  LIN {X 14334.988,Y 2494.793,Z -328.660,A -89.99654,B 0.00000,C 180.00000} ; insert
  LIN {X 14334.988,Y 2494.793,Z -328.660,A -89.99654,B 0.00000,C 180.00000} ; release
  LIN {X 14334.988,Y 2494.793,Z -28.660,A -89.99654,B 0.00000,C 180.00000} ; retreat
  ; Step 1131, bar 1482
  LIN {X 14434.988,Y 2494.793,Z 907.454,A -89.99654,B 0.00000,C 180.00000} ; outside
  LIN {X 14434.988,Y 2494.793,Z -78.660,A -89.99654,B 0.00000,C 180.00000} ; preinsert
  LIN {X 14434.988,Y 2494.793,Z -328.660,A -89.99654,B 0.00000,C 180.00000} ; insert
  LIN {X 14434.988,Y 2494.793,Z -328.660,A -89.99654,B 0.00000,C 180.00000} ; release
  LIN {X 14434.988,Y 2494.793,Z -28.660,A -89.99654,B 0.00000,C 180.00000} ; retreat
  ; Step 1132, bar 1484
  LIN {X 14534.988,Y 2494.793,Z 907.454,A -89.99654,B 0.00000,C 180.00000} ; outside
  LIN {X 14534.988,Y 2494.793,Z -78.660,A -89.99654,B 0.00000,C 180.00000} ; preinsert
  LIN {X 14534.988,Y 2494.793,Z -328.660,A -89.99654,B 0.00000,C 180.00000} ; insert
  LIN {X 14534.988,Y 2494.793,Z -328.660,A -89.99654,B 0.00000,C 180.00000} ; release
  LIN {X 14534.988,Y 2494.793,Z -28.660,A -89.99654,B 0.00000,C 180.00000} ; retreat
  ; Step 1133, bar 1486
  LIN {X 14634.988,Y 2494.793,Z 907.454,A -89.99654,B 0.00000,C 180.00000} ; outside
  LIN {X 14634.988,Y 2494.793,Z -78.660,A -89.99654,B 0.00000,C 180.00000} ; preinsert
  LIN {X 14634.988,Y 2494.793,Z -328.660,A -89.99654,B 0.00000,C 180.00000} ; insert
  LIN {X 14634.988,Y 2494.793,Z -328.660,A -89.99654,B 0.00000,C 180.00000} ; release
  LIN {X 14634.988,Y 2494.793,Z -28.660,A -89.99654,B 0.00000,C 180.00000} ; retreat
  ; Step 1134, bar 1488
  LIN {X 14734.988,Y 2494.793,Z 907.454,A -89.99654,B 0.00000,C 180.00000} ; outside
  LIN {X 14734.988,Y 2494.793,Z -78.660,A -89.99654,B 0.00000,C 180.00000} ; preinsert
  LIN {X 14734.988,Y 2494.793,Z -328.660,A -89.99654,B 0.00000,C 180.00000} ; insert
  LIN {X 14734.988,Y 2494.793,Z -328.660,A -89.99654,B 0.00000,C 180.00000} ; release
  LIN {X 14734.988,Y 2494.793,Z -28.660,A -89.99654,B 0.00000,C 180.00000} ; retreat
  ; Step 1135, bar 1490
  LIN {X 14834.988,Y 2494.793,Z 907.454,A -89.99654,B 0.00000,C 180.00000} ; outside
  LIN {X 14834.988,Y 2494.793,Z -78.660,A -89.99654,B 0.00000,C 180.00000} ; preinsert
  LIN {X 14834.988,Y 2494.793,Z -328.660,A -89.99654,B 0.00000,C 180.00000} ; insert
  LIN {X 14834.988,Y 2494.793,Z -328.660,A -89.99654,B 0.00000,C 180.00000} ; release
  LIN {X 14834.988,Y 2494.793,Z -28.660,A -89.99654,B 0.00000,C 180.00000} ; retreat
  ; Step 1136, bar 1492
  LIN {X 14934.988,Y 2494.793,Z 907.454,A -89.99654,B 0.00000,C 180.00000} ; outside
  LIN {X 14934.988,Y 2494.793,Z -78.660,A -89.99654,B 0.00000,C 180.00000} ; preinsert
  LIN {X 14934.988,Y 2494.793,Z -328.660,A -89.99654,B 0.00000,C 180.00000} ; insert
  LIN {X 14934.988,Y 2494.793,Z -328.660,A -89.99654,B 0.00000,C 180.00000} ; release
  LIN {X 14934.988,Y 2494.793,Z -28.660,A -89.99654,B 0.00000,C 180.00000} ; retreat
  ; Step 1137, bar 1494
  LIN {X 15034.988,Y 2494.793,Z 907.454,A -89.99654,B 0.00000,C 180.00000} ; outside
  LIN {X 15034.988,Y 2494.793,Z -78.660,A -89.99654,B 0.00000,C 180.00000} ; preinsert
  LIN {X 15034.988,Y 2494.793,Z -328.660,A -89.99654,B 0.00000,C 180.00000} ; insert
  LIN {X 15034.988,Y 2494.793,Z -328.660,A -89.99654,B 0.00000,C 180.00000} ; release
  LIN {X 15034.988,Y 2494.793,Z -28.660,A -89.99654,B 0.00000,C 180.00000} ; retreat
  ; Step 1138, bar 1496
  LIN {X 15134.988,Y 2494.793,Z 907.454,A -89.99654,B 0.00000,C 180.00000} ; outside
  LIN {X 15134.988,Y 2494.793,Z -78.660,A -89.99654,B 0.00000,C 180.00000} ; preinsert
  LIN {X 15134.988,Y 2494.793,Z -328.660,A -89.99654,B 0.00000,C 180.00000} ; insert
  LIN {X 15134.988,Y 2494.793,Z -328.660,A -89.99654,B 0.00000,C 180.00000} ; release
  LIN {X 15134.988,Y 2494.793,Z -28.660,A -89.99654,B 0.00000,C 180.00000} ; retreat
  ; Step 1139, bar 1498
  LIN {X 15234.988,Y 2494.793,Z 907.454,A -89.99654,B 0.00000,C 180.00000} ; outside
  LIN {X 15234.988,Y 2494.793,Z -78.660,A -89.99654,B 0.00000,C 180.00000} ; preinsert
  LIN {X 15234.988,Y 2494.793,Z -328.660,A -89.99654,B 0.00000,C 180.00000} ; insert
  LIN {X 15234.988,Y 2494.793,Z -328.660,A -89.99654,B 0.00000,C 180.00000} ; release
  LIN {X 15234.988,Y 2494.793,Z -28.660,A -89.99654,B 0.00000,C 180.00000} ; retreat
  ; Step 1140, bar 1500
  LIN {X 15334.988,Y 2494.793,Z 907.454,A -89.99654,B 0.00000,C 180.00000} ; outside
  LIN {X 15334.988,Y 2494.793,Z -78.660,A -89.99654,B 0.00000,C 180.00000} ; preinsert
  LIN {X 15334.988,Y 2494.793,Z -328.660,A -89.99654,B 0.00000,C 180.00000} ; insert
  LIN {X 15334.988,Y 2494.793,Z -328.660,A -89.99654,B 0.00000,C 180.00000} ; release
  LIN {X 15334.988,Y 2494.793,Z -28.660,A -89.99654,B 0.00000,C 180.00000} ; retreat
  ; Step 1141, bar 1502
  LIN {X 15434.988,Y 2494.793,Z 907.454,A -89.99654,B 0.00000,C 180.00000} ; outside
  LIN {X 15434.988,Y 2494.793,Z -78.660,A -89.99654,B 0.00000,C 180.00000} ; preinsert
  LIN {X 15434.988,Y 2494.793,Z -328.660,A -89.99654,B 0.00000,C 180.00000} ; insert
  LIN {X 15434.988,Y 2494.793,Z -328.660,A -89.99654,B 0.00000,C 180.00000} ; release
  LIN {X 15434.988,Y 2494.793,Z -28.660,A -89.99654,B 0.00000,C 180.00000} ; retreat
  ; Step 1142, bar 1504
  LIN {X 15534.988,Y 2494.793,Z 907.454,A -89.99654,B 0.00000,C 180.00000} ; outside
  LIN {X 15534.988,Y 2494.793,Z -78.660,A -89.99654,B 0.00000,C 180.00000} ; preinsert
  LIN {X 15534.988,Y 2494.793,Z -328.660,A -89.99654,B 0.00000,C 180.00000} ; insert
  LIN {X 15534.988,Y 2494.793,Z -328.660,A -89.99654,B 0.00000,C 180.00000} ; release
  LIN {X 15534.988,Y 2494.793,Z -28.660,A -89.99654,B 0.00000,C 180.00000} ; retreat
  ; Step 1143, bar 1506
  LIN {X 15634.988,Y 2494.793,Z 907.454,A -89.99654,B 0.00000,C 180.00000} ; outside
  LIN {X 15634.988,Y 2494.793,Z -78.660,A -89.99654,B 0.00000,C 180.00000} ; preinsert
  LIN {X 15634.988,Y 2494.793,Z -328.660,A -89.99654,B 0.00000,C 180.00000} ; insert
  LIN {X 15634.988,Y 2494.793,Z -328.660,A -89.99654,B 0.00000,C 180.00000} ; release
  LIN {X 15634.988,Y 2494.793,Z -28.660,A -89.99654,B 0.00000,C 180.00000} ; retreat
  ; Step 1144, bar 1508
  LIN {X 15734.988,Y 2494.793,Z 907.454,A -89.99654,B 0.00000,C 180.00000} ; outside
  LIN {X 15734.988,Y 2494.793,Z -78.660,A -89.99654,B 0.00000,C 180.00000} ; preinsert
  LIN {X 15734.988,Y 2494.793,Z -328.660,A -89.99654,B 0.00000,C 180.00000} ; insert
  LIN {X 15734.988,Y 2494.793,Z -328.660,A -89.99654,B 0.00000,C 180.00000} ; release
  LIN {X 15734.988,Y 2494.793,Z -28.660,A -89.99654,B 0.00000,C 180.00000} ; retreat
  ; Step 1145, bar 1510
  LIN {X 15834.988,Y 2494.793,Z 907.454,A -89.99654,B 0.00000,C 180.00000} ; outside
  LIN {X 15834.988,Y 2494.793,Z -78.660,A -89.99654,B 0.00000,C 180.00000} ; preinsert
  LIN {X 15834.988,Y 2494.793,Z -328.660,A -89.99654,B 0.00000,C 180.00000} ; insert
  LIN {X 15834.988,Y 2494.793,Z -328.660,A -89.99654,B 0.00000,C 180.00000} ; release
  LIN {X 15834.988,Y 2494.793,Z -28.660,A -89.99654,B 0.00000,C 180.00000} ; retreat
  ; Step 1146, bar 1512
  LIN {X 15934.988,Y 2494.793,Z 907.454,A -89.99654,B 0.00000,C 180.00000} ; outside
  LIN {X 15934.988,Y 2494.793,Z -78.660,A -89.99654,B 0.00000,C 180.00000} ; preinsert
  LIN {X 15934.988,Y 2494.793,Z -328.660,A -89.99654,B 0.00000,C 180.00000} ; insert
  LIN {X 15934.988,Y 2494.793,Z -328.660,A -89.99654,B 0.00000,C 180.00000} ; release
  LIN {X 15934.988,Y 2494.793,Z -28.660,A -89.99654,B 0.00000,C 180.00000} ; retreat
  ; Step 1147, bar 1514
  LIN {X 16034.988,Y 2494.793,Z 907.454,A -89.99654,B 0.00000,C 180.00000} ; outside
  LIN {X 16034.988,Y 2494.793,Z -78.660,A -89.99654,B 0.00000,C 180.00000} ; preinsert
  LIN {X 16034.988,Y 2494.793,Z -328.660,A -89.99654,B 0.00000,C 180.00000} ; insert
  LIN {X 16034.988,Y 2494.793,Z -328.660,A -89.99654,B 0.00000,C 180.00000} ; release
  LIN {X 16034.988,Y 2494.793,Z -28.660,A -89.99654,B 0.00000,C 180.00000} ; retreat
  ; Step 1148, bar 1807
  LIN {X -14334.988,Y -2494.793,Z 907.454,A 90.00346,B 0.00000,C 180.00000} ; outside
  LIN {X -14334.988,Y -2494.793,Z -78.660,A 90.00346,B 0.00000,C 180.00000} ; preinsert
  LIN {X -14334.988,Y -2494.793,Z -328.660,A 90.00346,B 0.00000,C 180.00000} ; insert
  LIN {X -14334.988,Y -2494.793,Z -328.660,A 90.00346,B 0.00000,C 180.00000} ; release
  LIN {X -14334.988,Y -2494.793,Z -28.660,A 90.00346,B 0.00000,C 180.00000} ; retreat
  ; Step 1149, bar 1809
  LIN {X -14434.988,Y -2494.793,Z 907.454,A 90.00346,B 0.00000,C 180.00000} ; outside
  LIN {X -14434.988,Y -2494.793,Z -78.660,A 90.00346,B 0.00000,C 180.00000} ; preinsert
  LIN {X -14434.988,Y -2494.793,Z -328.660,A 90.00346,B 0.00000,C 180.00000} ; insert
  LIN {X -14434.988,Y -2494.793,Z -328.660,A 90.00346,B 0.00000,C 180.00000} ; release
  LIN {X -14434.988,Y -2494.793,Z -28.660,A 90.00346,B 0.00000,C 180.00000} ; retreat
  ; Step 1150, bar 1811
  LIN {X -14534.988,Y -2494.793,Z 907.454,A 90.00346,B 0.00000,C 180.00000} ; outside
  LIN {X -14534.988,Y -2494.793,Z -78.660,A 90.00346,B 0.00000,C 180.00000} ; preinsert
  LIN {X -14534.988,Y -2494.793,Z -328.660,A 90.00346,B 0.00000,C 180.00000} ; insert
  LIN {X -14534.988,Y -2494.793,Z -328.660,A 90.00346,B 0.00000,C 180.00000} ; release
  LIN {X -14534.988,Y -2494.793,Z -28.660,A 90.00346,B 0.00000,C 180.00000} ; retreat
  ; Step 1151, bar 1813
  LIN {X -14634.988,Y -2494.793,Z 907.454,A 90.00346,B 0.00000,C 180.00000} ; outside
  LIN {X -14634.988,Y -2494.793,Z -78.660,A 90.00346,B 0.00000,C 180.00000} ; preinsert
  LIN {X -14634.988,Y -2494.793,Z -328.660,A 90.00346,B 0.00000,C 180.00000} ; insert
  LIN {X -14634.988,Y -2494.793,Z -328.660,A 90.00346,B 0.00000,C 180.00000} ; release
  LIN {X -14634.988,Y -2494.793,Z -28.660,A 90.00346,B 0.00000,C 180.00000} ; retreat
  ; Step 1152, bar 1815
  LIN {X -14734.988,Y -2494.793,Z 907.454,A 90.00346,B 0.00000,C 180.00000} ; outside
  LIN {X -14734.988,Y -2494.793,Z -78.660,A 90.00346,B 0.00000,C 180.00000} ; preinsert
  LIN {X -14734.988,Y -2494.793,Z -328.660,A 90.00346,B 0.00000,C 180.00000} ; insert
  LIN {X -14734.988,Y -2494.793,Z -328.660,A 90.00346,B 0.00000,C 180.00000} ; release
  LIN {X -14734.988,Y -2494.793,Z -28.660,A 90.00346,B 0.00000,C 180.00000} ; retreat
  ; Step 1153, bar 1817
  LIN {X -14834.988,Y -2494.793,Z 907.454,A 90.00346,B 0.00000,C 180.00000} ; outside
  LIN {X -14834.988,Y -2494.793,Z -78.660,A 90.00346,B 0.00000,C 180.00000} ; preinsert
  LIN {X -14834.988,Y -2494.793,Z -328.660,A 90.00346,B 0.00000,C 180.00000} ; insert
  LIN {X -14834.988,Y -2494.793,Z -328.660,A 90.00346,B 0.00000,C 180.00000} ; release
  LIN {X -14834.988,Y -2494.793,Z -28.660,A 90.00346,B 0.00000,C 180.00000} ; retreat
  ; Step 1154, bar 1819
  LIN {X -14934.988,Y -2494.793,Z 907.454,A 90.00346,B 0.00000,C 180.00000} ; outside
  LIN {X -14934.988,Y -2494.793,Z -78.660,A 90.00346,B 0.00000,C 180.00000} ; preinsert
  LIN {X -14934.988,Y -2494.793,Z -328.660,A 90.00346,B 0.00000,C 180.00000} ; insert
  LIN {X -14934.988,Y -2494.793,Z -328.660,A 90.00346,B 0.00000,C 180.00000} ; release
  LIN {X -14934.988,Y -2494.793,Z -28.660,A 90.00346,B 0.00000,C 180.00000} ; retreat
  ; Step 1155, bar 1821
  LIN {X -15034.988,Y -2494.793,Z 907.454,A 90.00346,B 0.00000,C 180.00000} ; outside
  LIN {X -15034.988,Y -2494.793,Z -78.660,A 90.00346,B 0.00000,C 180.00000} ; preinsert
  LIN {X -15034.988,Y -2494.793,Z -328.660,A 90.00346,B 0.00000,C 180.00000} ; insert
  LIN {X -15034.988,Y -2494.793,Z -328.660,A 90.00346,B 0.00000,C 180.00000} ; release
  LIN {X -15034.988,Y -2494.793,Z -28.660,A 90.00346,B 0.00000,C 180.00000} ; retreat
  ; Step 1156, bar 1823
  LIN {X -15134.988,Y -2494.793,Z 907.454,A 90.00346,B 0.00000,C 180.00000} ; outside
  LIN {X -15134.988,Y -2494.793,Z -78.660,A 90.00346,B 0.00000,C 180.00000} ; preinsert
  LIN {X -15134.988,Y -2494.793,Z -328.660,A 90.00346,B 0.00000,C 180.00000} ; insert
  LIN {X -15134.988,Y -2494.793,Z -328.660,A 90.00346,B 0.00000,C 180.00000} ; release
  LIN {X -15134.988,Y -2494.793,Z -28.660,A 90.00346,B 0.00000,C 180.00000} ; retreat
  ; Step 1157, bar 1825
  LIN {X -15234.988,Y -2494.793,Z 907.454,A 90.00346,B 0.00000,C 180.00000} ; outside
  LIN {X -15234.988,Y -2494.793,Z -78.660,A 90.00346,B 0.00000,C 180.00000} ; preinsert
  LIN {X -15234.988,Y -2494.793,Z -328.660,A 90.00346,B 0.00000,C 180.00000} ; insert
  LIN {X -15234.988,Y -2494.793,Z -328.660,A 90.00346,B 0.00000,C 180.00000} ; release
  LIN {X -15234.988,Y -2494.793,Z -28.660,A 90.00346,B 0.00000,C 180.00000} ; retreat
  ; Step 1158, bar 1829
  LIN {X -15434.988,Y -2494.793,Z 907.454,A 90.00346,B 0.00000,C 180.00000} ; outside
  LIN {X -15434.988,Y -2494.793,Z -78.660,A 90.00346,B 0.00000,C 180.00000} ; preinsert
  LIN {X -15434.988,Y -2494.793,Z -328.660,A 90.00346,B 0.00000,C 180.00000} ; insert
  LIN {X -15434.988,Y -2494.793,Z -328.660,A 90.00346,B 0.00000,C 180.00000} ; release
  LIN {X -15434.988,Y -2494.793,Z -28.660,A 90.00346,B 0.00000,C 180.00000} ; retreat
  ; Step 1159, bar 1827
  LIN {X -15334.988,Y -2494.793,Z 907.454,A 90.00346,B 0.00000,C 180.00000} ; outside
  LIN {X -15334.988,Y -2494.793,Z -78.660,A 90.00346,B 0.00000,C 180.00000} ; preinsert
  LIN {X -15334.988,Y -2494.793,Z -328.660,A 90.00346,B 0.00000,C 180.00000} ; insert
  LIN {X -15334.988,Y -2494.793,Z -328.660,A 90.00346,B 0.00000,C 180.00000} ; release
  LIN {X -15334.988,Y -2494.793,Z -28.660,A 90.00346,B 0.00000,C 180.00000} ; retreat
  ; Step 1160, bar 1831
  LIN {X -15534.988,Y -2494.793,Z 907.454,A 90.00346,B 0.00000,C 180.00000} ; outside
  LIN {X -15534.988,Y -2494.793,Z -78.660,A 90.00346,B 0.00000,C 180.00000} ; preinsert
  LIN {X -15534.988,Y -2494.793,Z -328.660,A 90.00346,B 0.00000,C 180.00000} ; insert
  LIN {X -15534.988,Y -2494.793,Z -328.660,A 90.00346,B 0.00000,C 180.00000} ; release
  LIN {X -15534.988,Y -2494.793,Z -28.660,A 90.00346,B 0.00000,C 180.00000} ; retreat
  ; Step 1161, bar 1833
  LIN {X -15634.988,Y -2494.793,Z 907.454,A 90.00346,B 0.00000,C 180.00000} ; outside
  LIN {X -15634.988,Y -2494.793,Z -78.660,A 90.00346,B 0.00000,C 180.00000} ; preinsert
  LIN {X -15634.988,Y -2494.793,Z -328.660,A 90.00346,B 0.00000,C 180.00000} ; insert
  LIN {X -15634.988,Y -2494.793,Z -328.660,A 90.00346,B 0.00000,C 180.00000} ; release
  LIN {X -15634.988,Y -2494.793,Z -28.660,A 90.00346,B 0.00000,C 180.00000} ; retreat
  ; Step 1162, bar 1835
  LIN {X -15734.988,Y -2494.793,Z 907.454,A 90.00346,B 0.00000,C 180.00000} ; outside
  LIN {X -15734.988,Y -2494.793,Z -78.660,A 90.00346,B 0.00000,C 180.00000} ; preinsert
  LIN {X -15734.988,Y -2494.793,Z -328.660,A 90.00346,B 0.00000,C 180.00000} ; insert
  LIN {X -15734.988,Y -2494.793,Z -328.660,A 90.00346,B 0.00000,C 180.00000} ; release
  LIN {X -15734.988,Y -2494.793,Z -28.660,A 90.00346,B 0.00000,C 180.00000} ; retreat
  ; Step 1163, bar 1837
  LIN {X -15834.988,Y -2494.793,Z 907.454,A 90.00346,B 0.00000,C 180.00000} ; outside
  LIN {X -15834.988,Y -2494.793,Z -78.660,A 90.00346,B 0.00000,C 180.00000} ; preinsert
  LIN {X -15834.988,Y -2494.793,Z -328.660,A 90.00346,B 0.00000,C 180.00000} ; insert
  LIN {X -15834.988,Y -2494.793,Z -328.660,A 90.00346,B 0.00000,C 180.00000} ; release
  LIN {X -15834.988,Y -2494.793,Z -28.660,A 90.00346,B 0.00000,C 180.00000} ; retreat
  ; Step 1164, bar 1839
  LIN {X -15934.988,Y -2494.793,Z 907.454,A 90.00346,B 0.00000,C 180.00000} ; outside
  LIN {X -15934.988,Y -2494.793,Z -78.660,A 90.00346,B 0.00000,C 180.00000} ; preinsert
  LIN {X -15934.988,Y -2494.793,Z -328.660,A 90.00346,B 0.00000,C 180.00000} ; insert
  LIN {X -15934.988,Y -2494.793,Z -328.660,A 90.00346,B 0.00000,C 180.00000} ; release
  LIN {X -15934.988,Y -2494.793,Z -28.660,A 90.00346,B 0.00000,C 180.00000} ; retreat
  ; Step 1165, bar 1841
  LIN {X -16034.988,Y -2494.793,Z 907.454,A 90.00346,B 0.00000,C 180.00000} ; outside
  LIN {X -16034.988,Y -2494.793,Z -78.660,A 90.00346,B 0.00000,C 180.00000} ; preinsert
  LIN {X -16034.988,Y -2494.793,Z -328.660,A 90.00346,B 0.00000,C 180.00000} ; insert
  LIN {X -16034.988,Y -2494.793,Z -328.660,A 90.00346,B 0.00000,C 180.00000} ; release
  LIN {X -16034.988,Y -2494.793,Z -28.660,A 90.00346,B 0.00000,C 180.00000} ; retreat
  ; Step 1166, bar 1479
  LIN {X 14334.988,Y -2494.793,Z 907.454,A 89.99654,B 0.00000,C -180.00000} ; outside
  LIN {X 14334.988,Y -2494.793,Z -78.660,A 89.99654,B 0.00000,C -180.00000} ; preinsert
  LIN {X 14334.988,Y -2494.793,Z -328.660,A 89.99654,B 0.00000,C -180.00000} ; insert
  LIN {X 14334.988,Y -2494.793,Z -328.660,A 89.99654,B 0.00000,C -180.00000} ; release
  LIN {X 14334.988,Y -2494.793,Z -28.660,A 89.99654,B 0.00000,C -180.00000} ; retreat
  ; Step 1167, bar 1481
  LIN {X 14434.988,Y -2494.793,Z 907.454,A 89.99654,B 0.00000,C -180.00000} ; outside
  LIN {X 14434.988,Y -2494.793,Z -78.660,A 89.99654,B 0.00000,C -180.00000} ; preinsert
  LIN {X 14434.988,Y -2494.793,Z -328.660,A 89.99654,B 0.00000,C -180.00000} ; insert
  LIN {X 14434.988,Y -2494.793,Z -328.660,A 89.99654,B 0.00000,C -180.00000} ; release
  LIN {X 14434.988,Y -2494.793,Z -28.660,A 89.99654,B 0.00000,C -180.00000} ; retreat
  ; Step 1168, bar 1483
  LIN {X 14534.988,Y -2494.793,Z 907.454,A 89.99654,B 0.00000,C -180.00000} ; outside
  LIN {X 14534.988,Y -2494.793,Z -78.660,A 89.99654,B 0.00000,C -180.00000} ; preinsert
  LIN {X 14534.988,Y -2494.793,Z -328.660,A 89.99654,B 0.00000,C -180.00000} ; insert
  LIN {X 14534.988,Y -2494.793,Z -328.660,A 89.99654,B 0.00000,C -180.00000} ; release
  LIN {X 14534.988,Y -2494.793,Z -28.660,A 89.99654,B 0.00000,C -180.00000} ; retreat
  ; Step 1169, bar 1485
  LIN {X 14634.988,Y -2494.793,Z 907.454,A 89.99654,B 0.00000,C -180.00000} ; outside
  LIN {X 14634.988,Y -2494.793,Z -78.660,A 89.99654,B 0.00000,C -180.00000} ; preinsert
  LIN {X 14634.988,Y -2494.793,Z -328.660,A 89.99654,B 0.00000,C -180.00000} ; insert
  LIN {X 14634.988,Y -2494.793,Z -328.660,A 89.99654,B 0.00000,C -180.00000} ; release
  LIN {X 14634.988,Y -2494.793,Z -28.660,A 89.99654,B 0.00000,C -180.00000} ; retreat
  ; Step 1170, bar 1487
  LIN {X 14734.988,Y -2494.793,Z 907.454,A 89.99654,B 0.00000,C -180.00000} ; outside
  LIN {X 14734.988,Y -2494.793,Z -78.660,A 89.99654,B 0.00000,C -180.00000} ; preinsert
  LIN {X 14734.988,Y -2494.793,Z -328.660,A 89.99654,B 0.00000,C -180.00000} ; insert
  LIN {X 14734.988,Y -2494.793,Z -328.660,A 89.99654,B 0.00000,C -180.00000} ; release
  LIN {X 14734.988,Y -2494.793,Z -28.660,A 89.99654,B 0.00000,C -180.00000} ; retreat
  ; Step 1171, bar 1489
  LIN {X 14834.988,Y -2494.793,Z 907.454,A 89.99654,B 0.00000,C -180.00000} ; outside
  LIN {X 14834.988,Y -2494.793,Z -78.660,A 89.99654,B 0.00000,C -180.00000} ; preinsert
  LIN {X 14834.988,Y -2494.793,Z -328.660,A 89.99654,B 0.00000,C -180.00000} ; insert
  LIN {X 14834.988,Y -2494.793,Z -328.660,A 89.99654,B 0.00000,C -180.00000} ; release
  LIN {X 14834.988,Y -2494.793,Z -28.660,A 89.99654,B 0.00000,C -180.00000} ; retreat
  ; Step 1172, bar 1491
  LIN {X 14934.988,Y -2494.793,Z 907.454,A 89.99654,B 0.00000,C -180.00000} ; outside
  LIN {X 14934.988,Y -2494.793,Z -78.660,A 89.99654,B 0.00000,C -180.00000} ; preinsert
  LIN {X 14934.988,Y -2494.793,Z -328.660,A 89.99654,B 0.00000,C -180.00000} ; insert
  LIN {X 14934.988,Y -2494.793,Z -328.660,A 89.99654,B 0.00000,C -180.00000} ; release
  LIN {X 14934.988,Y -2494.793,Z -28.660,A 89.99654,B 0.00000,C -180.00000} ; retreat
  ; Step 1173, bar 1493
  LIN {X 15034.988,Y -2494.793,Z 907.454,A 89.99654,B 0.00000,C -180.00000} ; outside
  LIN {X 15034.988,Y -2494.793,Z -78.660,A 89.99654,B 0.00000,C -180.00000} ; preinsert
  LIN {X 15034.988,Y -2494.793,Z -328.660,A 89.99654,B 0.00000,C -180.00000} ; insert
  LIN {X 15034.988,Y -2494.793,Z -328.660,A 89.99654,B 0.00000,C -180.00000} ; release
  LIN {X 15034.988,Y -2494.793,Z -28.660,A 89.99654,B 0.00000,C -180.00000} ; retreat
  ; Step 1174, bar 1495
  LIN {X 15134.988,Y -2494.793,Z 907.454,A 89.99654,B 0.00000,C -180.00000} ; outside
  LIN {X 15134.988,Y -2494.793,Z -78.660,A 89.99654,B 0.00000,C -180.00000} ; preinsert
  LIN {X 15134.988,Y -2494.793,Z -328.660,A 89.99654,B 0.00000,C -180.00000} ; insert
  LIN {X 15134.988,Y -2494.793,Z -328.660,A 89.99654,B 0.00000,C -180.00000} ; release
  LIN {X 15134.988,Y -2494.793,Z -28.660,A 89.99654,B 0.00000,C -180.00000} ; retreat
  ; Step 1175, bar 1497
  LIN {X 15234.988,Y -2494.793,Z 907.454,A 89.99654,B 0.00000,C -180.00000} ; outside
  LIN {X 15234.988,Y -2494.793,Z -78.660,A 89.99654,B 0.00000,C -180.00000} ; preinsert
  LIN {X 15234.988,Y -2494.793,Z -328.660,A 89.99654,B 0.00000,C -180.00000} ; insert
  LIN {X 15234.988,Y -2494.793,Z -328.660,A 89.99654,B 0.00000,C -180.00000} ; release
  LIN {X 15234.988,Y -2494.793,Z -28.660,A 89.99654,B 0.00000,C -180.00000} ; retreat
  ; Step 1176, bar 1499
  LIN {X 15334.988,Y -2494.793,Z 907.454,A 89.99654,B 0.00000,C -180.00000} ; outside
  LIN {X 15334.988,Y -2494.793,Z -78.660,A 89.99654,B 0.00000,C -180.00000} ; preinsert
  LIN {X 15334.988,Y -2494.793,Z -328.660,A 89.99654,B 0.00000,C -180.00000} ; insert
  LIN {X 15334.988,Y -2494.793,Z -328.660,A 89.99654,B 0.00000,C -180.00000} ; release
  LIN {X 15334.988,Y -2494.793,Z -28.660,A 89.99654,B 0.00000,C -180.00000} ; retreat
  ; Step 1177, bar 1501
  LIN {X 15434.988,Y -2494.793,Z 907.454,A 89.99654,B 0.00000,C -180.00000} ; outside
  LIN {X 15434.988,Y -2494.793,Z -78.660,A 89.99654,B 0.00000,C -180.00000} ; preinsert
  LIN {X 15434.988,Y -2494.793,Z -328.660,A 89.99654,B 0.00000,C -180.00000} ; insert
  LIN {X 15434.988,Y -2494.793,Z -328.660,A 89.99654,B 0.00000,C -180.00000} ; release
  LIN {X 15434.988,Y -2494.793,Z -28.660,A 89.99654,B 0.00000,C -180.00000} ; retreat
  ; Step 1178, bar 1503
  LIN {X 15534.988,Y -2494.793,Z 907.454,A 89.99654,B 0.00000,C -180.00000} ; outside
  LIN {X 15534.988,Y -2494.793,Z -78.660,A 89.99654,B 0.00000,C -180.00000} ; preinsert
  LIN {X 15534.988,Y -2494.793,Z -328.660,A 89.99654,B 0.00000,C -180.00000} ; insert
  LIN {X 15534.988,Y -2494.793,Z -328.660,A 89.99654,B 0.00000,C -180.00000} ; release
  LIN {X 15534.988,Y -2494.793,Z -28.660,A 89.99654,B 0.00000,C -180.00000} ; retreat
  ; Step 1179, bar 1505
  LIN {X 15634.988,Y -2494.793,Z 907.454,A 89.99654,B 0.00000,C -180.00000} ; outside
  LIN {X 15634.988,Y -2494.793,Z -78.660,A 89.99654,B 0.00000,C -180.00000} ; preinsert
  LIN {X 15634.988,Y -2494.793,Z -328.660,A 89.99654,B 0.00000,C -180.00000} ; insert
  LIN {X 15634.988,Y -2494.793,Z -328.660,A 89.99654,B 0.00000,C -180.00000} ; release
  LIN {X 15634.988,Y -2494.793,Z -28.660,A 89.99654,B 0.00000,C -180.00000} ; retreat
  ; Step 1180, bar 1507
  LIN {X 15734.988,Y -2494.793,Z 907.454,A 89.99654,B 0.00000,C -180.00000} ; outside
  LIN {X 15734.988,Y -2494.793,Z -78.660,A 89.99654,B 0.00000,C -180.00000} ; preinsert
  LIN {X 15734.988,Y -2494.793,Z -328.660,A 89.99654,B 0.00000,C -180.00000} ; insert
  LIN {X 15734.988,Y -2494.793,Z -328.660,A 89.99654,B 0.00000,C -180.00000} ; release
  LIN {X 15734.988,Y -2494.793,Z -28.660,A 89.99654,B 0.00000,C -180.00000} ; retreat
  ; Step 1181, bar 1509
  LIN {X 15834.988,Y -2494.793,Z 907.454,A 89.99654,B 0.00000,C -180.00000} ; outside
  LIN {X 15834.988,Y -2494.793,Z -78.660,A 89.99654,B 0.00000,C -180.00000} ; preinsert
  LIN {X 15834.988,Y -2494.793,Z -328.660,A 89.99654,B 0.00000,C -180.00000} ; insert
  LIN {X 15834.988,Y -2494.793,Z -328.660,A 89.99654,B 0.00000,C -180.00000} ; release
  LIN {X 15834.988,Y -2494.793,Z -28.660,A 89.99654,B 0.00000,C -180.00000} ; retreat
  ; Step 1182, bar 1511
  LIN {X 15934.988,Y -2494.793,Z 907.454,A 89.99654,B 0.00000,C -180.00000} ; outside
  LIN {X 15934.988,Y -2494.793,Z -78.660,A 89.99654,B 0.00000,C -180.00000} ; preinsert
  LIN {X 15934.988,Y -2494.793,Z -328.660,A 89.99654,B 0.00000,C -180.00000} ; insert
  LIN {X 15934.988,Y -2494.793,Z -328.660,A 89.99654,B 0.00000,C -180.00000} ; release
  LIN {X 15934.988,Y -2494.793,Z -28.660,A 89.99654,B 0.00000,C -180.00000} ; retreat
  ; Step 1183, bar 1513
  LIN {X 16034.988,Y -2494.793,Z 907.454,A 89.99654,B 0.00000,C -180.00000} ; outside
  LIN {X 16034.988,Y -2494.793,Z -78.660,A 89.99654,B 0.00000,C -180.00000} ; preinsert
  LIN {X 16034.988,Y -2494.793,Z -328.660,A 89.99654,B 0.00000,C -180.00000} ; insert
  LIN {X 16034.988,Y -2494.793,Z -328.660,A 89.99654,B 0.00000,C -180.00000} ; release
  LIN {X 16034.988,Y -2494.793,Z -28.660,A 89.99654,B 0.00000,C -180.00000} ; retreat
  ; Step 1184, bar 1808
  LIN {X -14334.988,Y 2494.793,Z 907.454,A -90.00346,B 0.00000,C -180.00000} ; outside
  LIN {X -14334.988,Y 2494.793,Z -78.660,A -90.00346,B 0.00000,C -180.00000} ; preinsert
  LIN {X -14334.988,Y 2494.793,Z -328.660,A -90.00346,B 0.00000,C -180.00000} ; insert
  LIN {X -14334.988,Y 2494.793,Z -328.660,A -90.00346,B 0.00000,C -180.00000} ; release
  LIN {X -14334.988,Y 2494.793,Z -28.660,A -90.00346,B 0.00000,C -180.00000} ; retreat
  ; Step 1185, bar 1810
  LIN {X -14434.988,Y 2494.793,Z 907.454,A -90.00346,B 0.00000,C -180.00000} ; outside
  LIN {X -14434.988,Y 2494.793,Z -78.660,A -90.00346,B 0.00000,C -180.00000} ; preinsert
  LIN {X -14434.988,Y 2494.793,Z -328.660,A -90.00346,B 0.00000,C -180.00000} ; insert
  LIN {X -14434.988,Y 2494.793,Z -328.660,A -90.00346,B 0.00000,C -180.00000} ; release
  LIN {X -14434.988,Y 2494.793,Z -28.660,A -90.00346,B 0.00000,C -180.00000} ; retreat
  ; Step 1186, bar 1812
  LIN {X -14534.988,Y 2494.793,Z 907.454,A -90.00346,B 0.00000,C -180.00000} ; outside
  LIN {X -14534.988,Y 2494.793,Z -78.660,A -90.00346,B 0.00000,C -180.00000} ; preinsert
  LIN {X -14534.988,Y 2494.793,Z -328.660,A -90.00346,B 0.00000,C -180.00000} ; insert
  LIN {X -14534.988,Y 2494.793,Z -328.660,A -90.00346,B 0.00000,C -180.00000} ; release
  LIN {X -14534.988,Y 2494.793,Z -28.660,A -90.00346,B 0.00000,C -180.00000} ; retreat
  ; Step 1187, bar 1814
  LIN {X -14634.988,Y 2494.793,Z 907.454,A -90.00346,B 0.00000,C -180.00000} ; outside
  LIN {X -14634.988,Y 2494.793,Z -78.660,A -90.00346,B 0.00000,C -180.00000} ; preinsert
  LIN {X -14634.988,Y 2494.793,Z -328.660,A -90.00346,B 0.00000,C -180.00000} ; insert
  LIN {X -14634.988,Y 2494.793,Z -328.660,A -90.00346,B 0.00000,C -180.00000} ; release
  LIN {X -14634.988,Y 2494.793,Z -28.660,A -90.00346,B 0.00000,C -180.00000} ; retreat
  ; Step 1188, bar 1816
  LIN {X -14734.988,Y 2494.793,Z 907.454,A -90.00346,B 0.00000,C -180.00000} ; outside
  LIN {X -14734.988,Y 2494.793,Z -78.660,A -90.00346,B 0.00000,C -180.00000} ; preinsert
  LIN {X -14734.988,Y 2494.793,Z -328.660,A -90.00346,B 0.00000,C -180.00000} ; insert
  LIN {X -14734.988,Y 2494.793,Z -328.660,A -90.00346,B 0.00000,C -180.00000} ; release
  LIN {X -14734.988,Y 2494.793,Z -28.660,A -90.00346,B 0.00000,C -180.00000} ; retreat
  ; Step 1189, bar 1818
  LIN {X -14834.988,Y 2494.793,Z 907.454,A -90.00346,B 0.00000,C -180.00000} ; outside
  LIN {X -14834.988,Y 2494.793,Z -78.660,A -90.00346,B 0.00000,C -180.00000} ; preinsert
  LIN {X -14834.988,Y 2494.793,Z -328.660,A -90.00346,B 0.00000,C -180.00000} ; insert
  LIN {X -14834.988,Y 2494.793,Z -328.660,A -90.00346,B 0.00000,C -180.00000} ; release
  LIN {X -14834.988,Y 2494.793,Z -28.660,A -90.00346,B 0.00000,C -180.00000} ; retreat
  ; Step 1190, bar 1820
  LIN {X -14934.988,Y 2494.793,Z 907.454,A -90.00346,B 0.00000,C -180.00000} ; outside
  LIN {X -14934.988,Y 2494.793,Z -78.660,A -90.00346,B 0.00000,C -180.00000} ; preinsert
  LIN {X -14934.988,Y 2494.793,Z -328.660,A -90.00346,B 0.00000,C -180.00000} ; insert
  LIN {X -14934.988,Y 2494.793,Z -328.660,A -90.00346,B 0.00000,C -180.00000} ; release
  LIN {X -14934.988,Y 2494.793,Z -28.660,A -90.00346,B 0.00000,C -180.00000} ; retreat
  ; Step 1191, bar 1822
  LIN {X -15034.988,Y 2494.793,Z 907.454,A -90.00346,B 0.00000,C -180.00000} ; outside
  LIN {X -15034.988,Y 2494.793,Z -78.660,A -90.00346,B 0.00000,C -180.00000} ; preinsert
  LIN {X -15034.988,Y 2494.793,Z -328.660,A -90.00346,B 0.00000,C -180.00000} ; insert
  LIN {X -15034.988,Y 2494.793,Z -328.660,A -90.00346,B 0.00000,C -180.00000} ; release
  LIN {X -15034.988,Y 2494.793,Z -28.660,A -90.00346,B 0.00000,C -180.00000} ; retreat
  ; Step 1192, bar 1824
  LIN {X -15134.988,Y 2494.793,Z 907.454,A -90.00346,B 0.00000,C -180.00000} ; outside
  LIN {X -15134.988,Y 2494.793,Z -78.660,A -90.00346,B 0.00000,C -180.00000} ; preinsert
  LIN {X -15134.988,Y 2494.793,Z -328.660,A -90.00346,B 0.00000,C -180.00000} ; insert
  LIN {X -15134.988,Y 2494.793,Z -328.660,A -90.00346,B 0.00000,C -180.00000} ; release
  LIN {X -15134.988,Y 2494.793,Z -28.660,A -90.00346,B 0.00000,C -180.00000} ; retreat
  ; Step 1193, bar 1826
  LIN {X -15234.988,Y 2494.793,Z 907.454,A -90.00346,B 0.00000,C -180.00000} ; outside
  LIN {X -15234.988,Y 2494.793,Z -78.660,A -90.00346,B 0.00000,C -180.00000} ; preinsert
  LIN {X -15234.988,Y 2494.793,Z -328.660,A -90.00346,B 0.00000,C -180.00000} ; insert
  LIN {X -15234.988,Y 2494.793,Z -328.660,A -90.00346,B 0.00000,C -180.00000} ; release
  LIN {X -15234.988,Y 2494.793,Z -28.660,A -90.00346,B 0.00000,C -180.00000} ; retreat
  ; Step 1194, bar 1830
  LIN {X -15434.988,Y 2494.793,Z 907.454,A -90.00346,B 0.00000,C -180.00000} ; outside
  LIN {X -15434.988,Y 2494.793,Z -78.660,A -90.00346,B 0.00000,C -180.00000} ; preinsert
  LIN {X -15434.988,Y 2494.793,Z -328.660,A -90.00346,B 0.00000,C -180.00000} ; insert
  LIN {X -15434.988,Y 2494.793,Z -328.660,A -90.00346,B 0.00000,C -180.00000} ; release
  LIN {X -15434.988,Y 2494.793,Z -28.660,A -90.00346,B 0.00000,C -180.00000} ; retreat
  ; Step 1195, bar 1828
  LIN {X -15334.988,Y 2494.793,Z 907.454,A -90.00346,B 0.00000,C -180.00000} ; outside
  LIN {X -15334.988,Y 2494.793,Z -78.660,A -90.00346,B 0.00000,C -180.00000} ; preinsert
  LIN {X -15334.988,Y 2494.793,Z -328.660,A -90.00346,B 0.00000,C -180.00000} ; insert
  LIN {X -15334.988,Y 2494.793,Z -328.660,A -90.00346,B 0.00000,C -180.00000} ; release
  LIN {X -15334.988,Y 2494.793,Z -28.660,A -90.00346,B 0.00000,C -180.00000} ; retreat
  ; Step 1196, bar 1832
  LIN {X -15534.988,Y 2494.793,Z 907.454,A -90.00346,B 0.00000,C -180.00000} ; outside
  LIN {X -15534.988,Y 2494.793,Z -78.660,A -90.00346,B 0.00000,C -180.00000} ; preinsert
  LIN {X -15534.988,Y 2494.793,Z -328.660,A -90.00346,B 0.00000,C -180.00000} ; insert
  LIN {X -15534.988,Y 2494.793,Z -328.660,A -90.00346,B 0.00000,C -180.00000} ; release
  LIN {X -15534.988,Y 2494.793,Z -28.660,A -90.00346,B 0.00000,C -180.00000} ; retreat
  ; Step 1197, bar 1834
  LIN {X -15634.988,Y 2494.793,Z 907.454,A -90.00346,B 0.00000,C -180.00000} ; outside
  LIN {X -15634.988,Y 2494.793,Z -78.660,A -90.00346,B 0.00000,C -180.00000} ; preinsert
  LIN {X -15634.988,Y 2494.793,Z -328.660,A -90.00346,B 0.00000,C -180.00000} ; insert
  LIN {X -15634.988,Y 2494.793,Z -328.660,A -90.00346,B 0.00000,C -180.00000} ; release
  LIN {X -15634.988,Y 2494.793,Z -28.660,A -90.00346,B 0.00000,C -180.00000} ; retreat
  ; Step 1198, bar 1836
  LIN {X -15734.988,Y 2494.793,Z 907.454,A -90.00346,B 0.00000,C -180.00000} ; outside
  LIN {X -15734.988,Y 2494.793,Z -78.660,A -90.00346,B 0.00000,C -180.00000} ; preinsert
  LIN {X -15734.988,Y 2494.793,Z -328.660,A -90.00346,B 0.00000,C -180.00000} ; insert
  LIN {X -15734.988,Y 2494.793,Z -328.660,A -90.00346,B 0.00000,C -180.00000} ; release
  LIN {X -15734.988,Y 2494.793,Z -28.660,A -90.00346,B 0.00000,C -180.00000} ; retreat
  ; Step 1199, bar 1838
  LIN {X -15834.988,Y 2494.793,Z 907.454,A -90.00346,B 0.00000,C -180.00000} ; outside
  LIN {X -15834.988,Y 2494.793,Z -78.660,A -90.00346,B 0.00000,C -180.00000} ; preinsert
  LIN {X -15834.988,Y 2494.793,Z -328.660,A -90.00346,B 0.00000,C -180.00000} ; insert
  LIN {X -15834.988,Y 2494.793,Z -328.660,A -90.00346,B 0.00000,C -180.00000} ; release
  LIN {X -15834.988,Y 2494.793,Z -28.660,A -90.00346,B 0.00000,C -180.00000} ; retreat
  ; Step 1200, bar 1840
  LIN {X -15934.988,Y 2494.793,Z 907.454,A -90.00346,B 0.00000,C -180.00000} ; outside
  LIN {X -15934.988,Y 2494.793,Z -78.660,A -90.00346,B 0.00000,C -180.00000} ; preinsert
  LIN {X -15934.988,Y 2494.793,Z -328.660,A -90.00346,B 0.00000,C -180.00000} ; insert
  LIN {X -15934.988,Y 2494.793,Z -328.660,A -90.00346,B 0.00000,C -180.00000} ; release
  LIN {X -15934.988,Y 2494.793,Z -28.660,A -90.00346,B 0.00000,C -180.00000} ; retreat
  ; Step 1201, bar 1842
  LIN {X -16034.988,Y 2494.793,Z 907.454,A -90.00346,B 0.00000,C -180.00000} ; outside
  LIN {X -16034.988,Y 2494.793,Z -78.660,A -90.00346,B 0.00000,C -180.00000} ; preinsert
  LIN {X -16034.988,Y 2494.793,Z -328.660,A -90.00346,B 0.00000,C -180.00000} ; insert
  LIN {X -16034.988,Y 2494.793,Z -328.660,A -90.00346,B 0.00000,C -180.00000} ; release
  LIN {X -16034.988,Y 2494.793,Z -28.660,A -90.00346,B 0.00000,C -180.00000} ; retreat
  ; Step 1202, bar 1515
  LIN {X 16134.974,Y -2655.018,Z 888.947,A 90.01124,B 0.00000,C 180.00000} ; outside
  LIN {X 16134.974,Y -2655.018,Z -60.206,A 90.01124,B 0.00000,C 180.00000} ; preinsert
  LIN {X 16134.974,Y -2655.018,Z -310.206,A 90.01124,B 0.00000,C 180.00000} ; insert
  LIN {X 16134.974,Y -2655.018,Z -310.206,A 90.01124,B 0.00000,C 180.00000} ; release
  LIN {X 16134.974,Y -2655.018,Z -10.206,A 90.01124,B 0.00000,C 180.00000} ; retreat
  ; Step 1203, bar 1517
  LIN {X 16234.974,Y -2655.018,Z 888.947,A 90.01124,B 0.00000,C 180.00000} ; outside
  LIN {X 16234.974,Y -2655.018,Z -60.206,A 90.01124,B 0.00000,C 180.00000} ; preinsert
  LIN {X 16234.974,Y -2655.018,Z -310.206,A 90.01124,B 0.00000,C 180.00000} ; insert
  LIN {X 16234.974,Y -2655.018,Z -310.206,A 90.01124,B 0.00000,C 180.00000} ; release
  LIN {X 16234.974,Y -2655.018,Z -10.206,A 90.01124,B 0.00000,C 180.00000} ; retreat
  ; Step 1204, bar 1844
  LIN {X -16134.974,Y 2655.018,Z 888.947,A -89.98876,B 0.00000,C 180.00000} ; outside
  LIN {X -16134.974,Y 2655.018,Z -60.206,A -89.98876,B 0.00000,C 180.00000} ; preinsert
  LIN {X -16134.974,Y 2655.018,Z -310.206,A -89.98876,B 0.00000,C 180.00000} ; insert
  LIN {X -16134.974,Y 2655.018,Z -310.206,A -89.98876,B 0.00000,C 180.00000} ; release
  LIN {X -16134.974,Y 2655.018,Z -10.206,A -89.98876,B 0.00000,C 180.00000} ; retreat
  ; Step 1205, bar 1846
  LIN {X -16234.974,Y 2655.018,Z 888.947,A -89.98876,B 0.00000,C 180.00000} ; outside
  LIN {X -16234.974,Y 2655.018,Z -60.206,A -89.98876,B 0.00000,C 180.00000} ; preinsert
  LIN {X -16234.974,Y 2655.018,Z -310.206,A -89.98876,B 0.00000,C 180.00000} ; insert
  LIN {X -16234.974,Y 2655.018,Z -310.206,A -89.98876,B 0.00000,C 180.00000} ; release
  LIN {X -16234.974,Y 2655.018,Z -10.206,A -89.98876,B 0.00000,C 180.00000} ; retreat
  ; Step 1206, bar 1516
  LIN {X 16134.974,Y 2655.018,Z 888.947,A -90.01124,B 0.00000,C -180.00000} ; outside
  LIN {X 16134.974,Y 2655.018,Z -60.206,A -90.01124,B 0.00000,C -180.00000} ; preinsert
  LIN {X 16134.974,Y 2655.018,Z -310.206,A -90.01124,B 0.00000,C -180.00000} ; insert
  LIN {X 16134.974,Y 2655.018,Z -310.206,A -90.01124,B 0.00000,C -180.00000} ; release
  LIN {X 16134.974,Y 2655.018,Z -10.206,A -90.01124,B 0.00000,C -180.00000} ; retreat
  ; Step 1207, bar 1518
  LIN {X 16234.974,Y 2655.018,Z 888.947,A -90.01124,B 0.00000,C -180.00000} ; outside
  LIN {X 16234.974,Y 2655.018,Z -60.206,A -90.01124,B 0.00000,C -180.00000} ; preinsert
  LIN {X 16234.974,Y 2655.018,Z -310.206,A -90.01124,B 0.00000,C -180.00000} ; insert
  LIN {X 16234.974,Y 2655.018,Z -310.206,A -90.01124,B 0.00000,C -180.00000} ; release
  LIN {X 16234.974,Y 2655.018,Z -10.206,A -90.01124,B 0.00000,C -180.00000} ; retreat
  ; Step 1208, bar 1843
  LIN {X -16134.974,Y -2655.018,Z 888.947,A 89.98876,B 0.00000,C 180.00000} ; outside
  LIN {X -16134.974,Y -2655.018,Z -60.206,A 89.98876,B 0.00000,C 180.00000} ; preinsert
  LIN {X -16134.974,Y -2655.018,Z -310.206,A 89.98876,B 0.00000,C 180.00000} ; insert
  LIN {X -16134.974,Y -2655.018,Z -310.206,A 89.98876,B 0.00000,C 180.00000} ; release
  LIN {X -16134.974,Y -2655.018,Z -10.206,A 89.98876,B 0.00000,C 180.00000} ; retreat
  ; Step 1209, bar 1845
  LIN {X -16234.974,Y -2655.018,Z 888.947,A 89.98876,B 0.00000,C 180.00000} ; outside
  LIN {X -16234.974,Y -2655.018,Z -60.206,A 89.98876,B 0.00000,C 180.00000} ; preinsert
  LIN {X -16234.974,Y -2655.018,Z -310.206,A 89.98876,B 0.00000,C 180.00000} ; insert
  LIN {X -16234.974,Y -2655.018,Z -310.206,A 89.98876,B 0.00000,C 180.00000} ; release
  LIN {X -16234.974,Y -2655.018,Z -10.206,A 89.98876,B 0.00000,C 180.00000} ; retreat
  ; Step 1210, bar 1520
  LIN {X 1986.078,Y 2753.934,Z 892.365,A -89.99242,B 0.00000,C 180.00000} ; outside
  LIN {X 1986.078,Y 2753.934,Z -48.972,A -89.99242,B 0.00000,C 180.00000} ; preinsert
  LIN {X 1986.078,Y 2753.934,Z -298.972,A -89.99242,B 0.00000,C 180.00000} ; insert
  LIN {X 1986.078,Y 2753.934,Z -298.972,A -89.99242,B 0.00000,C 180.00000} ; release
  LIN {X 1986.078,Y 2753.934,Z 1.028,A -89.99242,B 0.00000,C 180.00000} ; retreat
  ; Step 1211, bar 1522
  LIN {X 5986.078,Y 2753.934,Z 892.365,A -89.99242,B 0.00000,C 180.00000} ; outside
  LIN {X 5986.078,Y 2753.934,Z -48.972,A -89.99242,B 0.00000,C 180.00000} ; preinsert
  LIN {X 5986.078,Y 2753.934,Z -298.972,A -89.99242,B 0.00000,C 180.00000} ; insert
  LIN {X 5986.078,Y 2753.934,Z -298.972,A -89.99242,B 0.00000,C 180.00000} ; release
  LIN {X 5986.078,Y 2753.934,Z 1.028,A -89.99242,B 0.00000,C 180.00000} ; retreat
  ; Step 1212, bar 1524
  LIN {X 9986.078,Y 2753.934,Z 892.365,A -89.99242,B 0.00000,C 180.00000} ; outside
  LIN {X 9986.078,Y 2753.934,Z -48.972,A -89.99242,B 0.00000,C 180.00000} ; preinsert
  LIN {X 9986.078,Y 2753.934,Z -298.972,A -89.99242,B 0.00000,C 180.00000} ; insert
  LIN {X 9986.078,Y 2753.934,Z -298.972,A -89.99242,B 0.00000,C 180.00000} ; release
  LIN {X 9986.078,Y 2753.934,Z 1.028,A -89.99242,B 0.00000,C 180.00000} ; retreat
  ; Step 1213, bar 1526
  LIN {X 13936.078,Y 2753.934,Z 892.365,A -89.99242,B 0.00000,C 180.00000} ; outside
  LIN {X 13936.078,Y 2753.934,Z -48.972,A -89.99242,B 0.00000,C 180.00000} ; preinsert
  LIN {X 13936.078,Y 2753.934,Z -298.972,A -89.99242,B 0.00000,C 180.00000} ; insert
  LIN {X 13936.078,Y 2753.934,Z -298.972,A -89.99242,B 0.00000,C 180.00000} ; release
  LIN {X 13936.078,Y 2753.934,Z 1.028,A -89.99242,B 0.00000,C 180.00000} ; retreat
  ; Step 1214, bar 1528
  LIN {X 14036.078,Y 2753.934,Z 892.365,A -89.99242,B 0.00000,C 180.00000} ; outside
  LIN {X 14036.078,Y 2753.934,Z -48.972,A -89.99242,B 0.00000,C 180.00000} ; preinsert
  LIN {X 14036.078,Y 2753.934,Z -298.972,A -89.99242,B 0.00000,C 180.00000} ; insert
  LIN {X 14036.078,Y 2753.934,Z -298.972,A -89.99242,B 0.00000,C 180.00000} ; release
  LIN {X 14036.078,Y 2753.934,Z 1.028,A -89.99242,B 0.00000,C 180.00000} ; retreat
  ; Step 1215, bar 1539
  LIN {X -1986.078,Y -2753.934,Z 892.365,A 90.00758,B 0.00000,C -180.00000} ; outside
  LIN {X -1986.078,Y -2753.934,Z -48.972,A 90.00758,B 0.00000,C -180.00000} ; preinsert
  LIN {X -1986.078,Y -2753.934,Z -298.972,A 90.00758,B 0.00000,C -180.00000} ; insert
  LIN {X -1986.078,Y -2753.934,Z -298.972,A 90.00758,B 0.00000,C -180.00000} ; release
  LIN {X -1986.078,Y -2753.934,Z 1.028,A 90.00758,B 0.00000,C -180.00000} ; retreat
  ; Step 1216, bar 1541
  LIN {X -5986.078,Y -2753.934,Z 892.365,A 90.00758,B 0.00000,C -180.00000} ; outside
  LIN {X -5986.078,Y -2753.934,Z -48.972,A 90.00758,B 0.00000,C -180.00000} ; preinsert
  LIN {X -5986.078,Y -2753.934,Z -298.972,A 90.00758,B 0.00000,C -180.00000} ; insert
  LIN {X -5986.078,Y -2753.934,Z -298.972,A 90.00758,B 0.00000,C -180.00000} ; release
  LIN {X -5986.078,Y -2753.934,Z 1.028,A 90.00758,B 0.00000,C -180.00000} ; retreat
  ; Step 1217, bar 1543
  LIN {X -9986.078,Y -2753.934,Z 892.365,A 90.00758,B 0.00000,C -180.00000} ; outside
  LIN {X -9986.078,Y -2753.934,Z -48.972,A 90.00758,B 0.00000,C -180.00000} ; preinsert
  LIN {X -9986.078,Y -2753.934,Z -298.972,A 90.00758,B 0.00000,C -180.00000} ; insert
  LIN {X -9986.078,Y -2753.934,Z -298.972,A 90.00758,B 0.00000,C -180.00000} ; release
  LIN {X -9986.078,Y -2753.934,Z 1.028,A 90.00758,B 0.00000,C -180.00000} ; retreat
  ; Step 1218, bar 1545
  LIN {X -13936.078,Y -2753.934,Z 892.365,A 90.00758,B 0.00000,C -180.00000} ; outside
  LIN {X -13936.078,Y -2753.934,Z -48.972,A 90.00758,B 0.00000,C -180.00000} ; preinsert
  LIN {X -13936.078,Y -2753.934,Z -298.972,A 90.00758,B 0.00000,C -180.00000} ; insert
  LIN {X -13936.078,Y -2753.934,Z -298.972,A 90.00758,B 0.00000,C -180.00000} ; release
  LIN {X -13936.078,Y -2753.934,Z 1.028,A 90.00758,B 0.00000,C -180.00000} ; retreat
  ; Step 1219, bar 1547
  LIN {X -14036.078,Y -2753.934,Z 892.365,A 90.00758,B 0.00000,C -180.00000} ; outside
  LIN {X -14036.078,Y -2753.934,Z -48.972,A 90.00758,B 0.00000,C -180.00000} ; preinsert
  LIN {X -14036.078,Y -2753.934,Z -298.972,A 90.00758,B 0.00000,C -180.00000} ; insert
  LIN {X -14036.078,Y -2753.934,Z -298.972,A 90.00758,B 0.00000,C -180.00000} ; release
  LIN {X -14036.078,Y -2753.934,Z 1.028,A 90.00758,B 0.00000,C -180.00000} ; retreat
  ; Step 1220, bar 1519
  LIN {X 1986.078,Y -2753.934,Z 892.365,A 89.99242,B 0.00000,C 180.00000} ; outside
  LIN {X 1986.078,Y -2753.934,Z -48.972,A 89.99242,B 0.00000,C 180.00000} ; preinsert
  LIN {X 1986.078,Y -2753.934,Z -298.972,A 89.99242,B 0.00000,C 180.00000} ; insert
  LIN {X 1986.078,Y -2753.934,Z -298.972,A 89.99242,B 0.00000,C 180.00000} ; release
  LIN {X 1986.078,Y -2753.934,Z 1.028,A 89.99242,B 0.00000,C 180.00000} ; retreat
  ; Step 1221, bar 1521
  LIN {X 5986.078,Y -2753.934,Z 892.365,A 89.99242,B 0.00000,C 180.00000} ; outside
  LIN {X 5986.078,Y -2753.934,Z -48.972,A 89.99242,B 0.00000,C 180.00000} ; preinsert
  LIN {X 5986.078,Y -2753.934,Z -298.972,A 89.99242,B 0.00000,C 180.00000} ; insert
  LIN {X 5986.078,Y -2753.934,Z -298.972,A 89.99242,B 0.00000,C 180.00000} ; release
  LIN {X 5986.078,Y -2753.934,Z 1.028,A 89.99242,B 0.00000,C 180.00000} ; retreat
  ; Step 1222, bar 1523
  LIN {X 9986.078,Y -2753.934,Z 892.365,A 89.99242,B 0.00000,C 180.00000} ; outside
  LIN {X 9986.078,Y -2753.934,Z -48.972,A 89.99242,B 0.00000,C 180.00000} ; preinsert
  LIN {X 9986.078,Y -2753.934,Z -298.972,A 89.99242,B 0.00000,C 180.00000} ; insert
  LIN {X 9986.078,Y -2753.934,Z -298.972,A 89.99242,B 0.00000,C 180.00000} ; release
  LIN {X 9986.078,Y -2753.934,Z 1.028,A 89.99242,B 0.00000,C 180.00000} ; retreat
  ; Step 1223, bar 1525
  LIN {X 13936.078,Y -2753.934,Z 892.365,A 89.99242,B 0.00000,C 180.00000} ; outside
  LIN {X 13936.078,Y -2753.934,Z -48.972,A 89.99242,B 0.00000,C 180.00000} ; preinsert
  LIN {X 13936.078,Y -2753.934,Z -298.972,A 89.99242,B 0.00000,C 180.00000} ; insert
  LIN {X 13936.078,Y -2753.934,Z -298.972,A 89.99242,B 0.00000,C 180.00000} ; release
  LIN {X 13936.078,Y -2753.934,Z 1.028,A 89.99242,B 0.00000,C 180.00000} ; retreat
  ; Step 1224, bar 1527
  LIN {X 14036.078,Y -2753.934,Z 892.365,A 89.99242,B 0.00000,C 180.00000} ; outside
  LIN {X 14036.078,Y -2753.934,Z -48.972,A 89.99242,B 0.00000,C 180.00000} ; preinsert
  LIN {X 14036.078,Y -2753.934,Z -298.972,A 89.99242,B 0.00000,C 180.00000} ; insert
  LIN {X 14036.078,Y -2753.934,Z -298.972,A 89.99242,B 0.00000,C 180.00000} ; release
  LIN {X 14036.078,Y -2753.934,Z 1.028,A 89.99242,B 0.00000,C 180.00000} ; retreat
  ; Step 1225, bar 1540
  LIN {X -1986.078,Y 2753.934,Z 892.365,A -90.00758,B 0.00000,C -180.00000} ; outside
  LIN {X -1986.078,Y 2753.934,Z -48.972,A -90.00758,B 0.00000,C -180.00000} ; preinsert
  LIN {X -1986.078,Y 2753.934,Z -298.972,A -90.00758,B 0.00000,C -180.00000} ; insert
  LIN {X -1986.078,Y 2753.934,Z -298.972,A -90.00758,B 0.00000,C -180.00000} ; release
  LIN {X -1986.078,Y 2753.934,Z 1.028,A -90.00758,B 0.00000,C -180.00000} ; retreat
  ; Step 1226, bar 1542
  LIN {X -5986.078,Y 2753.934,Z 892.365,A -90.00758,B 0.00000,C -180.00000} ; outside
  LIN {X -5986.078,Y 2753.934,Z -48.972,A -90.00758,B 0.00000,C -180.00000} ; preinsert
  LIN {X -5986.078,Y 2753.934,Z -298.972,A -90.00758,B 0.00000,C -180.00000} ; insert
  LIN {X -5986.078,Y 2753.934,Z -298.972,A -90.00758,B 0.00000,C -180.00000} ; release
  LIN {X -5986.078,Y 2753.934,Z 1.028,A -90.00758,B 0.00000,C -180.00000} ; retreat
  ; Step 1227, bar 1544
  LIN {X -9986.078,Y 2753.934,Z 892.365,A -90.00758,B 0.00000,C -180.00000} ; outside
  LIN {X -9986.078,Y 2753.934,Z -48.972,A -90.00758,B 0.00000,C -180.00000} ; preinsert
  LIN {X -9986.078,Y 2753.934,Z -298.972,A -90.00758,B 0.00000,C -180.00000} ; insert
  LIN {X -9986.078,Y 2753.934,Z -298.972,A -90.00758,B 0.00000,C -180.00000} ; release
  LIN {X -9986.078,Y 2753.934,Z 1.028,A -90.00758,B 0.00000,C -180.00000} ; retreat
  ; Step 1228, bar 1546
  LIN {X -13936.078,Y 2753.934,Z 892.365,A -90.00758,B 0.00000,C -180.00000} ; outside
  LIN {X -13936.078,Y 2753.934,Z -48.972,A -90.00758,B 0.00000,C -180.00000} ; preinsert
  LIN {X -13936.078,Y 2753.934,Z -298.972,A -90.00758,B 0.00000,C -180.00000} ; insert
  LIN {X -13936.078,Y 2753.934,Z -298.972,A -90.00758,B 0.00000,C -180.00000} ; release
  LIN {X -13936.078,Y 2753.934,Z 1.028,A -90.00758,B 0.00000,C -180.00000} ; retreat
  ; Step 1229, bar 1548
  LIN {X -14036.078,Y 2753.934,Z 892.365,A -90.00758,B 0.00000,C -180.00000} ; outside
  LIN {X -14036.078,Y 2753.934,Z -48.972,A -90.00758,B 0.00000,C -180.00000} ; preinsert
  LIN {X -14036.078,Y 2753.934,Z -298.972,A -90.00758,B 0.00000,C -180.00000} ; insert
  LIN {X -14036.078,Y 2753.934,Z -298.972,A -90.00758,B 0.00000,C -180.00000} ; release
  LIN {X -14036.078,Y 2753.934,Z 1.028,A -90.00758,B 0.00000,C -180.00000} ; retreat
  ; Step 1230, bar 2980
  LIN {X -12449.942,Y -1181.101,Z 1004.184,A 91.55051,B 0.00000,C 180.00000} ; outside
  LIN {X -12449.942,Y -1181.101,Z 62.437,A 91.55051,B 0.00000,C 180.00000} ; preinsert
  LIN {X -12449.942,Y -1181.101,Z -187.563,A 91.55051,B 0.00000,C 180.00000} ; insert
  LIN {X -12449.942,Y -1181.101,Z -187.563,A 91.55051,B 0.00000,C 180.00000} ; release
  LIN {X -12449.942,Y -1181.101,Z 112.437,A 91.55051,B 0.00000,C 180.00000} ; retreat
  ; Step 1231, bar 3019
  LIN {X 12449.942,Y -1181.101,Z 1004.184,A 88.44949,B 0.00000,C 180.00000} ; outside
  LIN {X 12449.942,Y -1181.101,Z 62.437,A 88.44949,B 0.00000,C 180.00000} ; preinsert
  LIN {X 12449.942,Y -1181.101,Z -187.563,A 88.44949,B 0.00000,C 180.00000} ; insert
  LIN {X 12449.942,Y -1181.101,Z -187.563,A 88.44949,B 0.00000,C 180.00000} ; release
  LIN {X 12449.942,Y -1181.101,Z 112.437,A 88.44949,B 0.00000,C 180.00000} ; retreat
  ; Step 1232, bar 2962
  LIN {X -12449.942,Y 1181.101,Z 1004.184,A -91.55051,B 0.00000,C -180.00000} ; outside
  LIN {X -12449.942,Y 1181.101,Z 62.437,A -91.55051,B 0.00000,C -180.00000} ; preinsert
  LIN {X -12449.942,Y 1181.101,Z -187.563,A -91.55051,B 0.00000,C -180.00000} ; insert
  LIN {X -12449.942,Y 1181.101,Z -187.563,A -91.55051,B 0.00000,C -180.00000} ; release
  LIN {X -12449.942,Y 1181.101,Z 112.437,A -91.55051,B 0.00000,C -180.00000} ; retreat
  ; Step 1233, bar 3001
  LIN {X 12449.942,Y 1181.101,Z 1004.184,A -88.44949,B 0.00000,C 180.00000} ; outside
  LIN {X 12449.942,Y 1181.101,Z 62.437,A -88.44949,B 0.00000,C 180.00000} ; preinsert
  LIN {X 12449.942,Y 1181.101,Z -187.563,A -88.44949,B 0.00000,C 180.00000} ; insert
  LIN {X 12449.942,Y 1181.101,Z -187.563,A -88.44949,B 0.00000,C 180.00000} ; release
  LIN {X 12449.942,Y 1181.101,Z 112.437,A -88.44949,B 0.00000,C 180.00000} ; retreat
  ; Step 1234, bar 279
  LIN {X 0.000,Y -125.000,Z 1131.871,A 0.00000,B 0.00000,C 180.00000} ; outside
  LIN {X 0.000,Y -125.000,Z 190.246,A 0.00000,B 0.00000,C 180.00000} ; preinsert
  LIN {X 0.000,Y -125.000,Z -59.754,A 0.00000,B 0.00000,C 180.00000} ; insert
  LIN {X 0.000,Y -125.000,Z -59.754,A 0.00000,B 0.00000,C 180.00000} ; release
  LIN {X 0.000,Y -125.000,Z 240.246,A 0.00000,B 0.00000,C 180.00000} ; retreat
  ; Step 1235, bar 306
  LIN {X 0.000,Y 125.000,Z 1131.871,A 0.00000,B 0.00000,C 180.00000} ; outside
  LIN {X 0.000,Y 125.000,Z 190.246,A 0.00000,B 0.00000,C 180.00000} ; preinsert
  LIN {X 0.000,Y 125.000,Z -59.754,A 0.00000,B 0.00000,C 180.00000} ; insert
  LIN {X 0.000,Y 125.000,Z -59.754,A 0.00000,B 0.00000,C 180.00000} ; release
  LIN {X 0.000,Y 125.000,Z 240.246,A 0.00000,B 0.00000,C 180.00000} ; retreat
  ; Step 1236, bar 1856
  LIN {X -15549.904,Y -1461.247,Z 792.807,A 89.99930,B 0.00000,C 180.00000} ; outside
  LIN {X -15549.904,Y -1461.247,Z -184.886,A 89.99930,B 0.00000,C 180.00000} ; preinsert
  LIN {X -15549.904,Y -1461.247,Z -434.886,A 89.99930,B 0.00000,C 180.00000} ; insert
  LIN {X -15549.904,Y -1461.247,Z -434.886,A 89.99930,B 0.00000,C 180.00000} ; release
  LIN {X -15549.904,Y -1461.247,Z -134.886,A 89.99930,B 0.00000,C 180.00000} ; retreat
  ; Step 1237, bar 1854
  LIN {X 15549.904,Y -1461.347,Z 792.807,A 90.00070,B 0.00000,C 180.00000} ; outside
  LIN {X 15549.904,Y -1461.347,Z -184.886,A 90.00070,B 0.00000,C 180.00000} ; preinsert
  LIN {X 15549.904,Y -1461.347,Z -434.886,A 90.00070,B 0.00000,C 180.00000} ; insert
  LIN {X 15549.904,Y -1461.347,Z -434.886,A 90.00070,B 0.00000,C 180.00000} ; release
  LIN {X 15549.904,Y -1461.347,Z -134.886,A 90.00070,B 0.00000,C 180.00000} ; retreat
  ; Step 1238, bar 1107
  LIN {X -15944.474,Y -1224.921,Z 793.619,A 0.02206,B 0.00000,C 180.00000} ; outside
  LIN {X -15944.474,Y -1224.921,Z -151.761,A 0.02206,B 0.00000,C 180.00000} ; preinsert
  LIN {X -15944.474,Y -1224.921,Z -401.761,A 0.02206,B 0.00000,C 180.00000} ; insert
  LIN {X -15944.474,Y -1224.921,Z -401.761,A 0.02206,B 0.00000,C 180.00000} ; release
  LIN {X -15944.474,Y -1224.921,Z -101.761,A 0.02206,B 0.00000,C 180.00000} ; retreat
  ; Step 1239, bar 1073
  LIN {X 15944.475,Y -1224.921,Z 793.619,A 179.97794,B 0.00000,C 180.00000} ; outside
  LIN {X 15944.475,Y -1224.921,Z -151.761,A 179.97794,B 0.00000,C 180.00000} ; preinsert
  LIN {X 15944.475,Y -1224.921,Z -401.761,A 179.97794,B 0.00000,C 180.00000} ; insert
  LIN {X 15944.475,Y -1224.921,Z -401.761,A 179.97794,B 0.00000,C 180.00000} ; release
  LIN {X 15944.475,Y -1224.921,Z -101.761,A 179.97794,B 0.00000,C 180.00000} ; retreat
  ; Step 1240, bar 1109
  LIN {X -15944.475,Y 1224.921,Z 793.619,A -0.02206,B 0.00000,C 180.00000} ; outside
  LIN {X -15944.475,Y 1224.921,Z -151.761,A -0.02206,B 0.00000,C 180.00000} ; preinsert
  LIN {X -15944.475,Y 1224.921,Z -401.761,A -0.02206,B 0.00000,C 180.00000} ; insert
  LIN {X -15944.475,Y 1224.921,Z -401.761,A -0.02206,B 0.00000,C 180.00000} ; release
  LIN {X -15944.475,Y 1224.921,Z -101.761,A -0.02206,B 0.00000,C 180.00000} ; retreat
  ; Step 1241, bar 1084
  LIN {X 15944.474,Y 1224.921,Z 793.619,A -179.97794,B 0.00000,C -180.00000} ; outside
  LIN {X 15944.474,Y 1224.921,Z -151.761,A -179.97794,B 0.00000,C -180.00000} ; preinsert
  LIN {X 15944.474,Y 1224.921,Z -401.761,A -179.97794,B 0.00000,C -180.00000} ; insert
  LIN {X 15944.474,Y 1224.921,Z -401.761,A -179.97794,B 0.00000,C -180.00000} ; release
  LIN {X 15944.474,Y 1224.921,Z -101.761,A -179.97794,B 0.00000,C -180.00000} ; retreat
  ; Step 1242, bar 1108
  LIN {X -15048.108,Y -1224.807,Z 804.035,A -179.98341,B 0.00000,C -180.00000} ; outside
  LIN {X -15048.108,Y -1224.807,Z -141.344,A -179.98341,B 0.00000,C -180.00000} ; preinsert
  LIN {X -15048.108,Y -1224.807,Z -391.344,A -179.98341,B 0.00000,C -180.00000} ; insert
  LIN {X -15048.108,Y -1224.807,Z -391.344,A -179.98341,B 0.00000,C -180.00000} ; release
  LIN {X -15048.108,Y -1224.807,Z -91.344,A -179.98341,B 0.00000,C -180.00000} ; retreat
  ; Step 1243, bar 1074
  LIN {X 15048.046,Y -1224.807,Z 804.038,A -0.01659,B 0.00000,C 180.00000} ; outside
  LIN {X 15048.046,Y -1224.807,Z -141.341,A -0.01659,B 0.00000,C 180.00000} ; preinsert
  LIN {X 15048.046,Y -1224.807,Z -391.341,A -0.01659,B 0.00000,C 180.00000} ; insert
  LIN {X 15048.046,Y -1224.807,Z -391.341,A -0.01659,B 0.00000,C 180.00000} ; release
  LIN {X 15048.046,Y -1224.807,Z -91.341,A -0.01659,B 0.00000,C 180.00000} ; retreat
  ; Step 1244, bar 1110
  LIN {X -15048.046,Y 1224.807,Z 804.038,A 179.98341,B 0.00000,C 180.00000} ; outside
  LIN {X -15048.046,Y 1224.807,Z -141.341,A 179.98341,B 0.00000,C 180.00000} ; preinsert
  LIN {X -15048.046,Y 1224.807,Z -391.341,A 179.98341,B 0.00000,C 180.00000} ; insert
  LIN {X -15048.046,Y 1224.807,Z -391.341,A 179.98341,B 0.00000,C 180.00000} ; release
  LIN {X -15048.046,Y 1224.807,Z -91.341,A 179.98341,B 0.00000,C 180.00000} ; retreat
  ; Step 1245, bar 1085
  LIN {X 15048.108,Y 1224.807,Z 804.035,A 0.01659,B 0.00000,C 180.00000} ; outside
  LIN {X 15048.108,Y 1224.807,Z -141.344,A 0.01659,B 0.00000,C 180.00000} ; preinsert
  LIN {X 15048.108,Y 1224.807,Z -391.344,A 0.01659,B 0.00000,C 180.00000} ; insert
  LIN {X 15048.108,Y 1224.807,Z -391.344,A 0.01659,B 0.00000,C 180.00000} ; release
  LIN {X 15048.108,Y 1224.807,Z -91.344,A 0.01659,B 0.00000,C 180.00000} ; retreat
  ; Step 1246, bar 2527
  LIN {X 16150.008,Y -2301.617,Z 992.570,A 89.15153,B 0.00000,C -180.00000} ; outside
  LIN {X 16150.008,Y -2301.617,Z 46.552,A 89.15153,B 0.00000,C -180.00000} ; preinsert
  LIN {X 16150.008,Y -2301.617,Z -203.448,A 89.15153,B 0.00000,C -180.00000} ; insert
  LIN {X 16150.008,Y -2301.617,Z -203.448,A 89.15153,B 0.00000,C -180.00000} ; release
  LIN {X 16150.008,Y -2301.617,Z 96.552,A 89.15153,B 0.00000,C -180.00000} ; retreat
  ; Step 1247, bar 2521
  LIN {X 15550.008,Y -2301.617,Z 992.570,A 89.15153,B 0.00000,C -180.00000} ; outside
  LIN {X 15550.008,Y -2301.617,Z 46.552,A 89.15153,B 0.00000,C -180.00000} ; preinsert
  LIN {X 15550.008,Y -2301.617,Z -203.448,A 89.15153,B 0.00000,C -180.00000} ; insert
  LIN {X 15550.008,Y -2301.617,Z -203.448,A 89.15153,B 0.00000,C -180.00000} ; release
  LIN {X 15550.008,Y -2301.617,Z 96.552,A 89.15153,B 0.00000,C -180.00000} ; retreat
  ; Step 1248, bar 2509
  LIN {X 14350.008,Y -2301.617,Z 992.570,A 89.15153,B 0.00000,C -180.00000} ; outside
  LIN {X 14350.008,Y -2301.617,Z 46.552,A 89.15153,B 0.00000,C -180.00000} ; preinsert
  LIN {X 14350.008,Y -2301.617,Z -203.448,A 89.15153,B 0.00000,C -180.00000} ; insert
  LIN {X 14350.008,Y -2301.617,Z -203.448,A 89.15153,B 0.00000,C -180.00000} ; release
  LIN {X 14350.008,Y -2301.617,Z 96.552,A 89.15153,B 0.00000,C -180.00000} ; retreat
  ; Step 1249, bar 2515
  LIN {X 14950.008,Y -2301.617,Z 992.570,A 89.15153,B 0.00000,C -180.00000} ; outside
  LIN {X 14950.008,Y -2301.617,Z 46.552,A 89.15153,B 0.00000,C -180.00000} ; preinsert
  LIN {X 14950.008,Y -2301.617,Z -203.448,A 89.15153,B 0.00000,C -180.00000} ; insert
  LIN {X 14950.008,Y -2301.617,Z -203.448,A 89.15153,B 0.00000,C -180.00000} ; release
  LIN {X 14950.008,Y -2301.617,Z 96.552,A 89.15153,B 0.00000,C -180.00000} ; retreat
  ; Step 1250, bar 2503
  LIN {X 13750.008,Y -2301.617,Z 992.570,A 89.15153,B 0.00000,C -180.00000} ; outside
  LIN {X 13750.008,Y -2301.617,Z 46.552,A 89.15153,B 0.00000,C -180.00000} ; preinsert
  LIN {X 13750.008,Y -2301.617,Z -203.448,A 89.15153,B 0.00000,C -180.00000} ; insert
  LIN {X 13750.008,Y -2301.617,Z -203.448,A 89.15153,B 0.00000,C -180.00000} ; release
  LIN {X 13750.008,Y -2301.617,Z 96.552,A 89.15153,B 0.00000,C -180.00000} ; retreat
  ; Step 1251, bar 2497
  LIN {X 13150.008,Y -2301.617,Z 992.570,A 89.15153,B 0.00000,C -180.00000} ; outside
  LIN {X 13150.008,Y -2301.617,Z 46.552,A 89.15153,B 0.00000,C -180.00000} ; preinsert
  LIN {X 13150.008,Y -2301.617,Z -203.448,A 89.15153,B 0.00000,C -180.00000} ; insert
  LIN {X 13150.008,Y -2301.617,Z -203.448,A 89.15153,B 0.00000,C -180.00000} ; release
  LIN {X 13150.008,Y -2301.617,Z 96.552,A 89.15153,B 0.00000,C -180.00000} ; retreat
  ; Step 1252, bar 2491
  LIN {X 12550.008,Y -2301.617,Z 992.570,A 89.15153,B 0.00000,C -180.00000} ; outside
  LIN {X 12550.008,Y -2301.617,Z 46.552,A 89.15153,B 0.00000,C -180.00000} ; preinsert
  LIN {X 12550.008,Y -2301.617,Z -203.448,A 89.15153,B 0.00000,C -180.00000} ; insert
  LIN {X 12550.008,Y -2301.617,Z -203.448,A 89.15153,B 0.00000,C -180.00000} ; release
  LIN {X 12550.008,Y -2301.617,Z 96.552,A 89.15153,B 0.00000,C -180.00000} ; retreat
  ; Step 1253, bar 2487
  LIN {X 12000.008,Y -2301.617,Z 992.570,A 89.15153,B 0.00000,C -180.00000} ; outside
  LIN {X 12000.008,Y -2301.617,Z 46.552,A 89.15153,B 0.00000,C -180.00000} ; preinsert
  LIN {X 12000.008,Y -2301.617,Z -203.448,A 89.15153,B 0.00000,C -180.00000} ; insert
  LIN {X 12000.008,Y -2301.617,Z -203.448,A 89.15153,B 0.00000,C -180.00000} ; release
  LIN {X 12000.008,Y -2301.617,Z 96.552,A 89.15153,B 0.00000,C -180.00000} ; retreat
  ; Step 1254, bar 2481
  LIN {X 11250.008,Y -2301.617,Z 992.570,A 89.15153,B 0.00000,C -180.00000} ; outside
  LIN {X 11250.008,Y -2301.617,Z 46.552,A 89.15153,B 0.00000,C -180.00000} ; preinsert
  LIN {X 11250.008,Y -2301.617,Z -203.448,A 89.15153,B 0.00000,C -180.00000} ; insert
  LIN {X 11250.008,Y -2301.617,Z -203.448,A 89.15153,B 0.00000,C -180.00000} ; release
  LIN {X 11250.008,Y -2301.617,Z 96.552,A 89.15153,B 0.00000,C -180.00000} ; retreat
  ; Step 1255, bar 2475
  LIN {X 10500.008,Y -2301.617,Z 992.570,A 89.15153,B 0.00000,C -180.00000} ; outside
  LIN {X 10500.008,Y -2301.617,Z 46.552,A 89.15153,B 0.00000,C -180.00000} ; preinsert
  LIN {X 10500.008,Y -2301.617,Z -203.448,A 89.15153,B 0.00000,C -180.00000} ; insert
  LIN {X 10500.008,Y -2301.617,Z -203.448,A 89.15153,B 0.00000,C -180.00000} ; release
  LIN {X 10500.008,Y -2301.617,Z 96.552,A 89.15153,B 0.00000,C -180.00000} ; retreat
  ; Step 1256, bar 2469
  LIN {X 9750.008,Y -2301.617,Z 992.570,A 89.15153,B 0.00000,C -180.00000} ; outside
  LIN {X 9750.008,Y -2301.617,Z 46.552,A 89.15153,B 0.00000,C -180.00000} ; preinsert
  LIN {X 9750.008,Y -2301.617,Z -203.448,A 89.15153,B 0.00000,C -180.00000} ; insert
  LIN {X 9750.008,Y -2301.617,Z -203.448,A 89.15153,B 0.00000,C -180.00000} ; release
  LIN {X 9750.008,Y -2301.617,Z 96.552,A 89.15153,B 0.00000,C -180.00000} ; retreat
  ; Step 1257, bar 2463
  LIN {X 9000.008,Y -2301.617,Z 992.570,A 89.15153,B 0.00000,C -180.00000} ; outside
  LIN {X 9000.008,Y -2301.617,Z 46.552,A 89.15153,B 0.00000,C -180.00000} ; preinsert
  LIN {X 9000.008,Y -2301.617,Z -203.448,A 89.15153,B 0.00000,C -180.00000} ; insert
  LIN {X 9000.008,Y -2301.617,Z -203.448,A 89.15153,B 0.00000,C -180.00000} ; release
  LIN {X 9000.008,Y -2301.617,Z 96.552,A 89.15153,B 0.00000,C -180.00000} ; retreat
  ; Step 1258, bar 2457
  LIN {X 8250.008,Y -2301.617,Z 992.570,A 89.15153,B 0.00000,C -180.00000} ; outside
  LIN {X 8250.008,Y -2301.617,Z 46.552,A 89.15153,B 0.00000,C -180.00000} ; preinsert
  LIN {X 8250.008,Y -2301.617,Z -203.448,A 89.15153,B 0.00000,C -180.00000} ; insert
  LIN {X 8250.008,Y -2301.617,Z -203.448,A 89.15153,B 0.00000,C -180.00000} ; release
  LIN {X 8250.008,Y -2301.617,Z 96.552,A 89.15153,B 0.00000,C -180.00000} ; retreat
  ; Step 1259, bar 2451
  LIN {X 7500.008,Y -2301.617,Z 992.570,A 89.15153,B 0.00000,C -180.00000} ; outside
  LIN {X 7500.008,Y -2301.617,Z 46.552,A 89.15153,B 0.00000,C -180.00000} ; preinsert
  LIN {X 7500.008,Y -2301.617,Z -203.448,A 89.15153,B 0.00000,C -180.00000} ; insert
  LIN {X 7500.008,Y -2301.617,Z -203.448,A 89.15153,B 0.00000,C -180.00000} ; release
  LIN {X 7500.008,Y -2301.617,Z 96.552,A 89.15153,B 0.00000,C -180.00000} ; retreat
  ; Step 1260, bar 2445
  LIN {X 6750.008,Y -2301.617,Z 992.570,A 89.15153,B 0.00000,C -180.00000} ; outside
  LIN {X 6750.008,Y -2301.617,Z 46.552,A 89.15153,B 0.00000,C -180.00000} ; preinsert
  LIN {X 6750.008,Y -2301.617,Z -203.448,A 89.15153,B 0.00000,C -180.00000} ; insert
  LIN {X 6750.008,Y -2301.617,Z -203.448,A 89.15153,B 0.00000,C -180.00000} ; release
  LIN {X 6750.008,Y -2301.617,Z 96.552,A 89.15153,B 0.00000,C -180.00000} ; retreat
  ; Step 1261, bar 2439
  LIN {X 6000.008,Y -2301.617,Z 992.570,A 89.15153,B 0.00000,C -180.00000} ; outside
  LIN {X 6000.008,Y -2301.617,Z 46.552,A 89.15153,B 0.00000,C -180.00000} ; preinsert
  LIN {X 6000.008,Y -2301.617,Z -203.448,A 89.15153,B 0.00000,C -180.00000} ; insert
  LIN {X 6000.008,Y -2301.617,Z -203.448,A 89.15153,B 0.00000,C -180.00000} ; release
  LIN {X 6000.008,Y -2301.617,Z 96.552,A 89.15153,B 0.00000,C -180.00000} ; retreat
  ; Step 1262, bar 2433
  LIN {X 5250.008,Y -2301.617,Z 992.570,A 89.15153,B 0.00000,C -180.00000} ; outside
  LIN {X 5250.008,Y -2301.617,Z 46.552,A 89.15153,B 0.00000,C -180.00000} ; preinsert
  LIN {X 5250.008,Y -2301.617,Z -203.448,A 89.15153,B 0.00000,C -180.00000} ; insert
  LIN {X 5250.008,Y -2301.617,Z -203.448,A 89.15153,B 0.00000,C -180.00000} ; release
  LIN {X 5250.008,Y -2301.617,Z 96.552,A 89.15153,B 0.00000,C -180.00000} ; retreat
  ; Step 1263, bar 2427
  LIN {X 4500.008,Y -2301.617,Z 992.570,A 89.15153,B 0.00000,C -180.00000} ; outside
  LIN {X 4500.008,Y -2301.617,Z 46.552,A 89.15153,B 0.00000,C -180.00000} ; preinsert
  LIN {X 4500.008,Y -2301.617,Z -203.448,A 89.15153,B 0.00000,C -180.00000} ; insert
  LIN {X 4500.008,Y -2301.617,Z -203.448,A 89.15153,B 0.00000,C -180.00000} ; release
  LIN {X 4500.008,Y -2301.617,Z 96.552,A 89.15153,B 0.00000,C -180.00000} ; retreat
  ; Step 1264, bar 2421
  LIN {X 3750.008,Y -2301.617,Z 992.570,A 89.15153,B 0.00000,C -180.00000} ; outside
  LIN {X 3750.008,Y -2301.617,Z 46.552,A 89.15153,B 0.00000,C -180.00000} ; preinsert
  LIN {X 3750.008,Y -2301.617,Z -203.448,A 89.15153,B 0.00000,C -180.00000} ; insert
  LIN {X 3750.008,Y -2301.617,Z -203.448,A 89.15153,B 0.00000,C -180.00000} ; release
  LIN {X 3750.008,Y -2301.617,Z 96.552,A 89.15153,B 0.00000,C -180.00000} ; retreat
  ; Step 1265, bar 2415
  LIN {X 3000.008,Y -2301.617,Z 992.570,A 89.15153,B 0.00000,C -180.00000} ; outside
  LIN {X 3000.008,Y -2301.617,Z 46.552,A 89.15153,B 0.00000,C -180.00000} ; preinsert
  LIN {X 3000.008,Y -2301.617,Z -203.448,A 89.15153,B 0.00000,C -180.00000} ; insert
  LIN {X 3000.008,Y -2301.617,Z -203.448,A 89.15153,B 0.00000,C -180.00000} ; release
  LIN {X 3000.008,Y -2301.617,Z 96.552,A 89.15153,B 0.00000,C -180.00000} ; retreat
  ; Step 1266, bar 2409
  LIN {X 2250.008,Y -2301.617,Z 992.570,A 89.15153,B 0.00000,C -180.00000} ; outside
  LIN {X 2250.008,Y -2301.617,Z 46.552,A 89.15153,B 0.00000,C -180.00000} ; preinsert
  LIN {X 2250.008,Y -2301.617,Z -203.448,A 89.15153,B 0.00000,C -180.00000} ; insert
  LIN {X 2250.008,Y -2301.617,Z -203.448,A 89.15153,B 0.00000,C -180.00000} ; release
  LIN {X 2250.008,Y -2301.617,Z 96.552,A 89.15153,B 0.00000,C -180.00000} ; retreat
  ; Step 1267, bar 2403
  LIN {X 1500.008,Y -2301.617,Z 992.570,A 89.15153,B 0.00000,C -180.00000} ; outside
  LIN {X 1500.008,Y -2301.617,Z 46.552,A 89.15153,B 0.00000,C -180.00000} ; preinsert
  LIN {X 1500.008,Y -2301.617,Z -203.448,A 89.15153,B 0.00000,C -180.00000} ; insert
  LIN {X 1500.008,Y -2301.617,Z -203.448,A 89.15153,B 0.00000,C -180.00000} ; release
  LIN {X 1500.008,Y -2301.617,Z 96.552,A 89.15153,B 0.00000,C -180.00000} ; retreat
  ; Step 1268, bar 2397
  LIN {X 750.008,Y -2301.617,Z 992.570,A 89.15153,B 0.00000,C 180.00000} ; outside
  LIN {X 750.008,Y -2301.617,Z 46.552,A 89.15153,B 0.00000,C 180.00000} ; preinsert
  LIN {X 750.008,Y -2301.617,Z -203.448,A 89.15153,B 0.00000,C 180.00000} ; insert
  LIN {X 750.008,Y -2301.617,Z -203.448,A 89.15153,B 0.00000,C 180.00000} ; release
  LIN {X 750.008,Y -2301.617,Z 96.552,A 89.15153,B 0.00000,C 180.00000} ; retreat
  ; Step 1269, bar 2253
  LIN {X -0.008,Y -2301.617,Z 992.570,A 90.84847,B 0.00000,C 180.00000} ; outside
  LIN {X -0.008,Y -2301.617,Z 46.552,A 90.84847,B 0.00000,C 180.00000} ; preinsert
  LIN {X -0.008,Y -2301.617,Z -203.448,A 90.84847,B 0.00000,C 180.00000} ; insert
  LIN {X -0.008,Y -2301.617,Z -203.448,A 90.84847,B 0.00000,C 180.00000} ; release
  LIN {X -0.008,Y -2301.617,Z 96.552,A 90.84847,B 0.00000,C 180.00000} ; retreat
  ; Step 1270, bar 2259
  LIN {X -750.008,Y -2301.617,Z 992.570,A 90.84847,B 0.00000,C 180.00000} ; outside
  LIN {X -750.008,Y -2301.617,Z 46.552,A 90.84847,B 0.00000,C 180.00000} ; preinsert
  LIN {X -750.008,Y -2301.617,Z -203.448,A 90.84847,B 0.00000,C 180.00000} ; insert
  LIN {X -750.008,Y -2301.617,Z -203.448,A 90.84847,B 0.00000,C 180.00000} ; release
  LIN {X -750.008,Y -2301.617,Z 96.552,A 90.84847,B 0.00000,C 180.00000} ; retreat
  ; Step 1271, bar 2265
  LIN {X -1500.008,Y -2301.617,Z 992.570,A 90.84847,B 0.00000,C 180.00000} ; outside
  LIN {X -1500.008,Y -2301.617,Z 46.552,A 90.84847,B 0.00000,C 180.00000} ; preinsert
  LIN {X -1500.008,Y -2301.617,Z -203.448,A 90.84847,B 0.00000,C 180.00000} ; insert
  LIN {X -1500.008,Y -2301.617,Z -203.448,A 90.84847,B 0.00000,C 180.00000} ; release
  LIN {X -1500.008,Y -2301.617,Z 96.552,A 90.84847,B 0.00000,C 180.00000} ; retreat
  ; Step 1272, bar 2271
  LIN {X -2250.008,Y -2301.617,Z 992.570,A 90.84847,B 0.00000,C 180.00000} ; outside
  LIN {X -2250.008,Y -2301.617,Z 46.552,A 90.84847,B 0.00000,C 180.00000} ; preinsert
  LIN {X -2250.008,Y -2301.617,Z -203.448,A 90.84847,B 0.00000,C 180.00000} ; insert
  LIN {X -2250.008,Y -2301.617,Z -203.448,A 90.84847,B 0.00000,C 180.00000} ; release
  LIN {X -2250.008,Y -2301.617,Z 96.552,A 90.84847,B 0.00000,C 180.00000} ; retreat
  ; Step 1273, bar 2277
  LIN {X -3000.008,Y -2301.617,Z 992.570,A 90.84847,B 0.00000,C 180.00000} ; outside
  LIN {X -3000.008,Y -2301.617,Z 46.552,A 90.84847,B 0.00000,C 180.00000} ; preinsert
  LIN {X -3000.008,Y -2301.617,Z -203.448,A 90.84847,B 0.00000,C 180.00000} ; insert
  LIN {X -3000.008,Y -2301.617,Z -203.448,A 90.84847,B 0.00000,C 180.00000} ; release
  LIN {X -3000.008,Y -2301.617,Z 96.552,A 90.84847,B 0.00000,C 180.00000} ; retreat
  ; Step 1274, bar 2283
  LIN {X -3750.008,Y -2301.617,Z 992.570,A 90.84847,B 0.00000,C 180.00000} ; outside
  LIN {X -3750.008,Y -2301.617,Z 46.552,A 90.84847,B 0.00000,C 180.00000} ; preinsert
  LIN {X -3750.008,Y -2301.617,Z -203.448,A 90.84847,B 0.00000,C 180.00000} ; insert
  LIN {X -3750.008,Y -2301.617,Z -203.448,A 90.84847,B 0.00000,C 180.00000} ; release
  LIN {X -3750.008,Y -2301.617,Z 96.552,A 90.84847,B 0.00000,C 180.00000} ; retreat
  ; Step 1275, bar 2289
  LIN {X -4500.008,Y -2301.617,Z 992.570,A 90.84847,B 0.00000,C 180.00000} ; outside
  LIN {X -4500.008,Y -2301.617,Z 46.552,A 90.84847,B 0.00000,C 180.00000} ; preinsert
  LIN {X -4500.008,Y -2301.617,Z -203.448,A 90.84847,B 0.00000,C 180.00000} ; insert
  LIN {X -4500.008,Y -2301.617,Z -203.448,A 90.84847,B 0.00000,C 180.00000} ; release
  LIN {X -4500.008,Y -2301.617,Z 96.552,A 90.84847,B 0.00000,C 180.00000} ; retreat
  ; Step 1276, bar 2295
  LIN {X -5250.008,Y -2301.617,Z 992.570,A 90.84847,B 0.00000,C 180.00000} ; outside
  LIN {X -5250.008,Y -2301.617,Z 46.552,A 90.84847,B 0.00000,C 180.00000} ; preinsert
  LIN {X -5250.008,Y -2301.617,Z -203.448,A 90.84847,B 0.00000,C 180.00000} ; insert
  LIN {X -5250.008,Y -2301.617,Z -203.448,A 90.84847,B 0.00000,C 180.00000} ; release
  LIN {X -5250.008,Y -2301.617,Z 96.552,A 90.84847,B 0.00000,C 180.00000} ; retreat
  ; Step 1277, bar 2301
  LIN {X -6000.008,Y -2301.617,Z 992.570,A 90.84847,B 0.00000,C 180.00000} ; outside
  LIN {X -6000.008,Y -2301.617,Z 46.552,A 90.84847,B 0.00000,C 180.00000} ; preinsert
  LIN {X -6000.008,Y -2301.617,Z -203.448,A 90.84847,B 0.00000,C 180.00000} ; insert
  LIN {X -6000.008,Y -2301.617,Z -203.448,A 90.84847,B 0.00000,C 180.00000} ; release
  LIN {X -6000.008,Y -2301.617,Z 96.552,A 90.84847,B 0.00000,C 180.00000} ; retreat
  ; Step 1278, bar 2307
  LIN {X -6750.008,Y -2301.617,Z 992.570,A 90.84847,B 0.00000,C 180.00000} ; outside
  LIN {X -6750.008,Y -2301.617,Z 46.552,A 90.84847,B 0.00000,C 180.00000} ; preinsert
  LIN {X -6750.008,Y -2301.617,Z -203.448,A 90.84847,B 0.00000,C 180.00000} ; insert
  LIN {X -6750.008,Y -2301.617,Z -203.448,A 90.84847,B 0.00000,C 180.00000} ; release
  LIN {X -6750.008,Y -2301.617,Z 96.552,A 90.84847,B 0.00000,C 180.00000} ; retreat
  ; Step 1279, bar 2313
  LIN {X -7500.008,Y -2301.617,Z 992.570,A 90.84847,B 0.00000,C 180.00000} ; outside
  LIN {X -7500.008,Y -2301.617,Z 46.552,A 90.84847,B 0.00000,C 180.00000} ; preinsert
  LIN {X -7500.008,Y -2301.617,Z -203.448,A 90.84847,B 0.00000,C 180.00000} ; insert
  LIN {X -7500.008,Y -2301.617,Z -203.448,A 90.84847,B 0.00000,C 180.00000} ; release
  LIN {X -7500.008,Y -2301.617,Z 96.552,A 90.84847,B 0.00000,C 180.00000} ; retreat
  ; Step 1280, bar 2319
  LIN {X -8250.008,Y -2301.617,Z 992.570,A 90.84847,B 0.00000,C 180.00000} ; outside
  LIN {X -8250.008,Y -2301.617,Z 46.552,A 90.84847,B 0.00000,C 180.00000} ; preinsert
  LIN {X -8250.008,Y -2301.617,Z -203.448,A 90.84847,B 0.00000,C 180.00000} ; insert
  LIN {X -8250.008,Y -2301.617,Z -203.448,A 90.84847,B 0.00000,C 180.00000} ; release
  LIN {X -8250.008,Y -2301.617,Z 96.552,A 90.84847,B 0.00000,C 180.00000} ; retreat
  ; Step 1281, bar 2325
  LIN {X -9000.008,Y -2301.617,Z 992.570,A 90.84847,B 0.00000,C 180.00000} ; outside
  LIN {X -9000.008,Y -2301.617,Z 46.552,A 90.84847,B 0.00000,C 180.00000} ; preinsert
  LIN {X -9000.008,Y -2301.617,Z -203.448,A 90.84847,B 0.00000,C 180.00000} ; insert
  LIN {X -9000.008,Y -2301.617,Z -203.448,A 90.84847,B 0.00000,C 180.00000} ; release
  LIN {X -9000.008,Y -2301.617,Z 96.552,A 90.84847,B 0.00000,C 180.00000} ; retreat
  ; Step 1282, bar 2331
  LIN {X -9750.008,Y -2301.617,Z 992.570,A 90.84847,B 0.00000,C 180.00000} ; outside
  LIN {X -9750.008,Y -2301.617,Z 46.552,A 90.84847,B 0.00000,C 180.00000} ; preinsert
  LIN {X -9750.008,Y -2301.617,Z -203.448,A 90.84847,B 0.00000,C 180.00000} ; insert
  LIN {X -9750.008,Y -2301.617,Z -203.448,A 90.84847,B 0.00000,C 180.00000} ; release
  LIN {X -9750.008,Y -2301.617,Z 96.552,A 90.84847,B 0.00000,C 180.00000} ; retreat
  ; Step 1283, bar 2337
  LIN {X -10500.008,Y -2301.617,Z 992.570,A 90.84847,B 0.00000,C 180.00000} ; outside
  LIN {X -10500.008,Y -2301.617,Z 46.552,A 90.84847,B 0.00000,C 180.00000} ; preinsert
  LIN {X -10500.008,Y -2301.617,Z -203.448,A 90.84847,B 0.00000,C 180.00000} ; insert
  LIN {X -10500.008,Y -2301.617,Z -203.448,A 90.84847,B 0.00000,C 180.00000} ; release
  LIN {X -10500.008,Y -2301.617,Z 96.552,A 90.84847,B 0.00000,C 180.00000} ; retreat
  ; Step 1284, bar 2343
  LIN {X -11250.008,Y -2301.617,Z 992.570,A 90.84847,B 0.00000,C 180.00000} ; outside
  LIN {X -11250.008,Y -2301.617,Z 46.552,A 90.84847,B 0.00000,C 180.00000} ; preinsert
  LIN {X -11250.008,Y -2301.617,Z -203.448,A 90.84847,B 0.00000,C 180.00000} ; insert
  LIN {X -11250.008,Y -2301.617,Z -203.448,A 90.84847,B 0.00000,C 180.00000} ; release
  LIN {X -11250.008,Y -2301.617,Z 96.552,A 90.84847,B 0.00000,C 180.00000} ; retreat
  ; Step 1285, bar 2349
  LIN {X -12000.008,Y -2301.617,Z 992.570,A 90.84847,B 0.00000,C 180.00000} ; outside
  LIN {X -12000.008,Y -2301.617,Z 46.552,A 90.84847,B 0.00000,C 180.00000} ; preinsert
  LIN {X -12000.008,Y -2301.617,Z -203.448,A 90.84847,B 0.00000,C 180.00000} ; insert
  LIN {X -12000.008,Y -2301.617,Z -203.448,A 90.84847,B 0.00000,C 180.00000} ; release
  LIN {X -12000.008,Y -2301.617,Z 96.552,A 90.84847,B 0.00000,C 180.00000} ; retreat
  ; Step 1286, bar 2353
  LIN {X -12550.008,Y -2301.617,Z 992.570,A 90.84847,B 0.00000,C 180.00000} ; outside
  LIN {X -12550.008,Y -2301.617,Z 46.552,A 90.84847,B 0.00000,C 180.00000} ; preinsert
  LIN {X -12550.008,Y -2301.617,Z -203.448,A 90.84847,B 0.00000,C 180.00000} ; insert
  LIN {X -12550.008,Y -2301.617,Z -203.448,A 90.84847,B 0.00000,C 180.00000} ; release
  LIN {X -12550.008,Y -2301.617,Z 96.552,A 90.84847,B 0.00000,C 180.00000} ; retreat
  ; Step 1287, bar 2359
  LIN {X -13150.008,Y -2301.617,Z 992.570,A 90.84847,B 0.00000,C 180.00000} ; outside
  LIN {X -13150.008,Y -2301.617,Z 46.552,A 90.84847,B 0.00000,C 180.00000} ; preinsert
  LIN {X -13150.008,Y -2301.617,Z -203.448,A 90.84847,B 0.00000,C 180.00000} ; insert
  LIN {X -13150.008,Y -2301.617,Z -203.448,A 90.84847,B 0.00000,C 180.00000} ; release
  LIN {X -13150.008,Y -2301.617,Z 96.552,A 90.84847,B 0.00000,C 180.00000} ; retreat
  ; Step 1288, bar 2365
  LIN {X -13750.008,Y -2301.617,Z 992.570,A 90.84847,B 0.00000,C 180.00000} ; outside
  LIN {X -13750.008,Y -2301.617,Z 46.552,A 90.84847,B 0.00000,C 180.00000} ; preinsert
  LIN {X -13750.008,Y -2301.617,Z -203.448,A 90.84847,B 0.00000,C 180.00000} ; insert
  LIN {X -13750.008,Y -2301.617,Z -203.448,A 90.84847,B 0.00000,C 180.00000} ; release
  LIN {X -13750.008,Y -2301.617,Z 96.552,A 90.84847,B 0.00000,C 180.00000} ; retreat
  ; Step 1289, bar 2377
  LIN {X -14950.008,Y -2301.617,Z 992.570,A 90.84847,B 0.00000,C 180.00000} ; outside
  LIN {X -14950.008,Y -2301.617,Z 46.552,A 90.84847,B 0.00000,C 180.00000} ; preinsert
  LIN {X -14950.008,Y -2301.617,Z -203.448,A 90.84847,B 0.00000,C 180.00000} ; insert
  LIN {X -14950.008,Y -2301.617,Z -203.448,A 90.84847,B 0.00000,C 180.00000} ; release
  LIN {X -14950.008,Y -2301.617,Z 96.552,A 90.84847,B 0.00000,C 180.00000} ; retreat
  ; Step 1290, bar 2371
  LIN {X -14350.008,Y -2301.617,Z 992.570,A 90.84847,B 0.00000,C 180.00000} ; outside
  LIN {X -14350.008,Y -2301.617,Z 46.552,A 90.84847,B 0.00000,C 180.00000} ; preinsert
  LIN {X -14350.008,Y -2301.617,Z -203.448,A 90.84847,B 0.00000,C 180.00000} ; insert
  LIN {X -14350.008,Y -2301.617,Z -203.448,A 90.84847,B 0.00000,C 180.00000} ; release
  LIN {X -14350.008,Y -2301.617,Z 96.552,A 90.84847,B 0.00000,C 180.00000} ; retreat
  ; Step 1291, bar 2383
  LIN {X -15550.008,Y -2301.617,Z 992.570,A 90.84847,B 0.00000,C 180.00000} ; outside
  LIN {X -15550.008,Y -2301.617,Z 46.552,A 90.84847,B 0.00000,C 180.00000} ; preinsert
  LIN {X -15550.008,Y -2301.617,Z -203.448,A 90.84847,B 0.00000,C 180.00000} ; insert
  LIN {X -15550.008,Y -2301.617,Z -203.448,A 90.84847,B 0.00000,C 180.00000} ; release
  LIN {X -15550.008,Y -2301.617,Z 96.552,A 90.84847,B 0.00000,C 180.00000} ; retreat
  ; Step 1292, bar 2389
  LIN {X -16150.008,Y -2301.617,Z 992.570,A 90.84847,B 0.00000,C 180.00000} ; outside
  LIN {X -16150.008,Y -2301.617,Z 46.552,A 90.84847,B 0.00000,C 180.00000} ; preinsert
  LIN {X -16150.008,Y -2301.617,Z -203.448,A 90.84847,B 0.00000,C 180.00000} ; insert
  LIN {X -16150.008,Y -2301.617,Z -203.448,A 90.84847,B 0.00000,C 180.00000} ; release
  LIN {X -16150.008,Y -2301.617,Z 96.552,A 90.84847,B 0.00000,C 180.00000} ; retreat
  ; Step 1293, bar 2110
  LIN {X -16150.008,Y 2301.617,Z 992.570,A -90.84847,B 0.00000,C -180.00000} ; outside
  LIN {X -16150.008,Y 2301.617,Z 46.552,A -90.84847,B 0.00000,C -180.00000} ; preinsert
  LIN {X -16150.008,Y 2301.617,Z -203.448,A -90.84847,B 0.00000,C -180.00000} ; insert
  LIN {X -16150.008,Y 2301.617,Z -203.448,A -90.84847,B 0.00000,C -180.00000} ; release
  LIN {X -16150.008,Y 2301.617,Z 96.552,A -90.84847,B 0.00000,C -180.00000} ; retreat
  ; Step 1294, bar 2104
  LIN {X -15550.008,Y 2301.617,Z 992.570,A -90.84847,B 0.00000,C -180.00000} ; outside
  LIN {X -15550.008,Y 2301.617,Z 46.552,A -90.84847,B 0.00000,C -180.00000} ; preinsert
  LIN {X -15550.008,Y 2301.617,Z -203.448,A -90.84847,B 0.00000,C -180.00000} ; insert
  LIN {X -15550.008,Y 2301.617,Z -203.448,A -90.84847,B 0.00000,C -180.00000} ; release
  LIN {X -15550.008,Y 2301.617,Z 96.552,A -90.84847,B 0.00000,C -180.00000} ; retreat
  ; Step 1295, bar 2098
  LIN {X -14950.008,Y 2301.617,Z 992.570,A -90.84847,B 0.00000,C -180.00000} ; outside
  LIN {X -14950.008,Y 2301.617,Z 46.552,A -90.84847,B 0.00000,C -180.00000} ; preinsert
  LIN {X -14950.008,Y 2301.617,Z -203.448,A -90.84847,B 0.00000,C -180.00000} ; insert
  LIN {X -14950.008,Y 2301.617,Z -203.448,A -90.84847,B 0.00000,C -180.00000} ; release
  LIN {X -14950.008,Y 2301.617,Z 96.552,A -90.84847,B 0.00000,C -180.00000} ; retreat
  ; Step 1296, bar 2092
  LIN {X -14350.008,Y 2301.617,Z 992.570,A -90.84847,B 0.00000,C -180.00000} ; outside
  LIN {X -14350.008,Y 2301.617,Z 46.552,A -90.84847,B 0.00000,C -180.00000} ; preinsert
  LIN {X -14350.008,Y 2301.617,Z -203.448,A -90.84847,B 0.00000,C -180.00000} ; insert
  LIN {X -14350.008,Y 2301.617,Z -203.448,A -90.84847,B 0.00000,C -180.00000} ; release
  LIN {X -14350.008,Y 2301.617,Z 96.552,A -90.84847,B 0.00000,C -180.00000} ; retreat
  ; Step 1297, bar 2086
  LIN {X -13750.008,Y 2301.617,Z 992.570,A -90.84847,B 0.00000,C -180.00000} ; outside
  LIN {X -13750.008,Y 2301.617,Z 46.552,A -90.84847,B 0.00000,C -180.00000} ; preinsert
  LIN {X -13750.008,Y 2301.617,Z -203.448,A -90.84847,B 0.00000,C -180.00000} ; insert
  LIN {X -13750.008,Y 2301.617,Z -203.448,A -90.84847,B 0.00000,C -180.00000} ; release
  LIN {X -13750.008,Y 2301.617,Z 96.552,A -90.84847,B 0.00000,C -180.00000} ; retreat
  ; Step 1298, bar 2080
  LIN {X -13150.008,Y 2301.617,Z 992.570,A -90.84847,B 0.00000,C -180.00000} ; outside
  LIN {X -13150.008,Y 2301.617,Z 46.552,A -90.84847,B 0.00000,C -180.00000} ; preinsert
  LIN {X -13150.008,Y 2301.617,Z -203.448,A -90.84847,B 0.00000,C -180.00000} ; insert
  LIN {X -13150.008,Y 2301.617,Z -203.448,A -90.84847,B 0.00000,C -180.00000} ; release
  LIN {X -13150.008,Y 2301.617,Z 96.552,A -90.84847,B 0.00000,C -180.00000} ; retreat
  ; Step 1299, bar 2074
  LIN {X -12550.008,Y 2301.617,Z 992.570,A -90.84847,B 0.00000,C -180.00000} ; outside
  LIN {X -12550.008,Y 2301.617,Z 46.552,A -90.84847,B 0.00000,C -180.00000} ; preinsert
  LIN {X -12550.008,Y 2301.617,Z -203.448,A -90.84847,B 0.00000,C -180.00000} ; insert
  LIN {X -12550.008,Y 2301.617,Z -203.448,A -90.84847,B 0.00000,C -180.00000} ; release
  LIN {X -12550.008,Y 2301.617,Z 96.552,A -90.84847,B 0.00000,C -180.00000} ; retreat
  ; Step 1300, bar 2070
  LIN {X -12000.008,Y 2301.617,Z 992.570,A -90.84847,B 0.00000,C -180.00000} ; outside
  LIN {X -12000.008,Y 2301.617,Z 46.552,A -90.84847,B 0.00000,C -180.00000} ; preinsert
  LIN {X -12000.008,Y 2301.617,Z -203.448,A -90.84847,B 0.00000,C -180.00000} ; insert
  LIN {X -12000.008,Y 2301.617,Z -203.448,A -90.84847,B 0.00000,C -180.00000} ; release
  LIN {X -12000.008,Y 2301.617,Z 96.552,A -90.84847,B 0.00000,C -180.00000} ; retreat
  ; Step 1301, bar 2064
  LIN {X -11250.008,Y 2301.617,Z 992.570,A -90.84847,B 0.00000,C -180.00000} ; outside
  LIN {X -11250.008,Y 2301.617,Z 46.552,A -90.84847,B 0.00000,C -180.00000} ; preinsert
  LIN {X -11250.008,Y 2301.617,Z -203.448,A -90.84847,B 0.00000,C -180.00000} ; insert
  LIN {X -11250.008,Y 2301.617,Z -203.448,A -90.84847,B 0.00000,C -180.00000} ; release
  LIN {X -11250.008,Y 2301.617,Z 96.552,A -90.84847,B 0.00000,C -180.00000} ; retreat
  ; Step 1302, bar 2058
  LIN {X -10500.008,Y 2301.617,Z 992.570,A -90.84847,B 0.00000,C -180.00000} ; outside
  LIN {X -10500.008,Y 2301.617,Z 46.552,A -90.84847,B 0.00000,C -180.00000} ; preinsert
  LIN {X -10500.008,Y 2301.617,Z -203.448,A -90.84847,B 0.00000,C -180.00000} ; insert
  LIN {X -10500.008,Y 2301.617,Z -203.448,A -90.84847,B 0.00000,C -180.00000} ; release
  LIN {X -10500.008,Y 2301.617,Z 96.552,A -90.84847,B 0.00000,C -180.00000} ; retreat
  ; Step 1303, bar 2052
  LIN {X -9750.008,Y 2301.617,Z 992.570,A -90.84847,B 0.00000,C -180.00000} ; outside
  LIN {X -9750.008,Y 2301.617,Z 46.552,A -90.84847,B 0.00000,C -180.00000} ; preinsert
  LIN {X -9750.008,Y 2301.617,Z -203.448,A -90.84847,B 0.00000,C -180.00000} ; insert
  LIN {X -9750.008,Y 2301.617,Z -203.448,A -90.84847,B 0.00000,C -180.00000} ; release
  LIN {X -9750.008,Y 2301.617,Z 96.552,A -90.84847,B 0.00000,C -180.00000} ; retreat
  ; Step 1304, bar 2046
  LIN {X -9000.008,Y 2301.617,Z 992.570,A -90.84847,B 0.00000,C -180.00000} ; outside
  LIN {X -9000.008,Y 2301.617,Z 46.552,A -90.84847,B 0.00000,C -180.00000} ; preinsert
  LIN {X -9000.008,Y 2301.617,Z -203.448,A -90.84847,B 0.00000,C -180.00000} ; insert
  LIN {X -9000.008,Y 2301.617,Z -203.448,A -90.84847,B 0.00000,C -180.00000} ; release
  LIN {X -9000.008,Y 2301.617,Z 96.552,A -90.84847,B 0.00000,C -180.00000} ; retreat
  ; Step 1305, bar 2040
  LIN {X -8250.008,Y 2301.617,Z 992.570,A -90.84847,B 0.00000,C -180.00000} ; outside
  LIN {X -8250.008,Y 2301.617,Z 46.552,A -90.84847,B 0.00000,C -180.00000} ; preinsert
  LIN {X -8250.008,Y 2301.617,Z -203.448,A -90.84847,B 0.00000,C -180.00000} ; insert
  LIN {X -8250.008,Y 2301.617,Z -203.448,A -90.84847,B 0.00000,C -180.00000} ; release
  LIN {X -8250.008,Y 2301.617,Z 96.552,A -90.84847,B 0.00000,C -180.00000} ; retreat
  ; Step 1306, bar 2034
  LIN {X -7500.008,Y 2301.617,Z 992.570,A -90.84847,B 0.00000,C -180.00000} ; outside
  LIN {X -7500.008,Y 2301.617,Z 46.552,A -90.84847,B 0.00000,C -180.00000} ; preinsert
  LIN {X -7500.008,Y 2301.617,Z -203.448,A -90.84847,B 0.00000,C -180.00000} ; insert
  LIN {X -7500.008,Y 2301.617,Z -203.448,A -90.84847,B 0.00000,C -180.00000} ; release
  LIN {X -7500.008,Y 2301.617,Z 96.552,A -90.84847,B 0.00000,C -180.00000} ; retreat
  ; Step 1307, bar 2028
  LIN {X -6750.008,Y 2301.617,Z 992.570,A -90.84847,B 0.00000,C -180.00000} ; outside
  LIN {X -6750.008,Y 2301.617,Z 46.552,A -90.84847,B 0.00000,C -180.00000} ; preinsert
  LIN {X -6750.008,Y 2301.617,Z -203.448,A -90.84847,B 0.00000,C -180.00000} ; insert
  LIN {X -6750.008,Y 2301.617,Z -203.448,A -90.84847,B 0.00000,C -180.00000} ; release
  LIN {X -6750.008,Y 2301.617,Z 96.552,A -90.84847,B 0.00000,C -180.00000} ; retreat
  ; Step 1308, bar 2022
  LIN {X -6000.008,Y 2301.617,Z 992.570,A -90.84847,B 0.00000,C -180.00000} ; outside
  LIN {X -6000.008,Y 2301.617,Z 46.552,A -90.84847,B 0.00000,C -180.00000} ; preinsert
  LIN {X -6000.008,Y 2301.617,Z -203.448,A -90.84847,B 0.00000,C -180.00000} ; insert
  LIN {X -6000.008,Y 2301.617,Z -203.448,A -90.84847,B 0.00000,C -180.00000} ; release
  LIN {X -6000.008,Y 2301.617,Z 96.552,A -90.84847,B 0.00000,C -180.00000} ; retreat
  ; Step 1309, bar 2016
  LIN {X -5250.008,Y 2301.617,Z 992.570,A -90.84847,B 0.00000,C -180.00000} ; outside
  LIN {X -5250.008,Y 2301.617,Z 46.552,A -90.84847,B 0.00000,C -180.00000} ; preinsert
  LIN {X -5250.008,Y 2301.617,Z -203.448,A -90.84847,B 0.00000,C -180.00000} ; insert
  LIN {X -5250.008,Y 2301.617,Z -203.448,A -90.84847,B 0.00000,C -180.00000} ; release
  LIN {X -5250.008,Y 2301.617,Z 96.552,A -90.84847,B 0.00000,C -180.00000} ; retreat
  ; Step 1310, bar 2010
  LIN {X -4500.008,Y 2301.617,Z 992.570,A -90.84847,B 0.00000,C -180.00000} ; outside
  LIN {X -4500.008,Y 2301.617,Z 46.552,A -90.84847,B 0.00000,C -180.00000} ; preinsert
  LIN {X -4500.008,Y 2301.617,Z -203.448,A -90.84847,B 0.00000,C -180.00000} ; insert
  LIN {X -4500.008,Y 2301.617,Z -203.448,A -90.84847,B 0.00000,C -180.00000} ; release
  LIN {X -4500.008,Y 2301.617,Z 96.552,A -90.84847,B 0.00000,C -180.00000} ; retreat
  ; Step 1311, bar 2004
  LIN {X -3750.008,Y 2301.617,Z 992.570,A -90.84847,B 0.00000,C -180.00000} ; outside
  LIN {X -3750.008,Y 2301.617,Z 46.552,A -90.84847,B 0.00000,C -180.00000} ; preinsert
  LIN {X -3750.008,Y 2301.617,Z -203.448,A -90.84847,B 0.00000,C -180.00000} ; insert
  LIN {X -3750.008,Y 2301.617,Z -203.448,A -90.84847,B 0.00000,C -180.00000} ; release
  LIN {X -3750.008,Y 2301.617,Z 96.552,A -90.84847,B 0.00000,C -180.00000} ; retreat
  ; Step 1312, bar 1998
  LIN {X -3000.008,Y 2301.617,Z 992.570,A -90.84847,B 0.00000,C -180.00000} ; outside
  LIN {X -3000.008,Y 2301.617,Z 46.552,A -90.84847,B 0.00000,C -180.00000} ; preinsert
  LIN {X -3000.008,Y 2301.617,Z -203.448,A -90.84847,B 0.00000,C -180.00000} ; insert
  LIN {X -3000.008,Y 2301.617,Z -203.448,A -90.84847,B 0.00000,C -180.00000} ; release
  LIN {X -3000.008,Y 2301.617,Z 96.552,A -90.84847,B 0.00000,C -180.00000} ; retreat
  ; Step 1313, bar 1992
  LIN {X -2250.008,Y 2301.617,Z 992.570,A -90.84847,B 0.00000,C -180.00000} ; outside
  LIN {X -2250.008,Y 2301.617,Z 46.552,A -90.84847,B 0.00000,C -180.00000} ; preinsert
  LIN {X -2250.008,Y 2301.617,Z -203.448,A -90.84847,B 0.00000,C -180.00000} ; insert
  LIN {X -2250.008,Y 2301.617,Z -203.448,A -90.84847,B 0.00000,C -180.00000} ; release
  LIN {X -2250.008,Y 2301.617,Z 96.552,A -90.84847,B 0.00000,C -180.00000} ; retreat
  ; Step 1314, bar 1986
  LIN {X -1500.008,Y 2301.617,Z 992.570,A -90.84847,B 0.00000,C -180.00000} ; outside
  LIN {X -1500.008,Y 2301.617,Z 46.552,A -90.84847,B 0.00000,C -180.00000} ; preinsert
  LIN {X -1500.008,Y 2301.617,Z -203.448,A -90.84847,B 0.00000,C -180.00000} ; insert
  LIN {X -1500.008,Y 2301.617,Z -203.448,A -90.84847,B 0.00000,C -180.00000} ; release
  LIN {X -1500.008,Y 2301.617,Z 96.552,A -90.84847,B 0.00000,C -180.00000} ; retreat
  ; Step 1315, bar 1980
  LIN {X -750.008,Y 2301.617,Z 992.570,A -90.84847,B 0.00000,C -180.00000} ; outside
  LIN {X -750.008,Y 2301.617,Z 46.552,A -90.84847,B 0.00000,C -180.00000} ; preinsert
  LIN {X -750.008,Y 2301.617,Z -203.448,A -90.84847,B 0.00000,C -180.00000} ; insert
  LIN {X -750.008,Y 2301.617,Z -203.448,A -90.84847,B 0.00000,C -180.00000} ; release
  LIN {X -750.008,Y 2301.617,Z 96.552,A -90.84847,B 0.00000,C -180.00000} ; retreat
  ; Step 1316, bar 1967
  LIN {X -0.008,Y 2301.617,Z 992.570,A -90.84847,B 0.00000,C -180.00000} ; outside
  LIN {X -0.008,Y 2301.617,Z 46.552,A -90.84847,B 0.00000,C -180.00000} ; preinsert
  LIN {X -0.008,Y 2301.617,Z -203.448,A -90.84847,B 0.00000,C -180.00000} ; insert
  LIN {X -0.008,Y 2301.617,Z -203.448,A -90.84847,B 0.00000,C -180.00000} ; release
  LIN {X -0.008,Y 2301.617,Z 96.552,A -90.84847,B 0.00000,C -180.00000} ; retreat
  ; Step 1317, bar 2118
  LIN {X 750.008,Y 2301.617,Z 992.570,A -89.15153,B 0.00000,C 180.00000} ; outside
  LIN {X 750.008,Y 2301.617,Z 46.552,A -89.15153,B 0.00000,C 180.00000} ; preinsert
  LIN {X 750.008,Y 2301.617,Z -203.448,A -89.15153,B 0.00000,C 180.00000} ; insert
  LIN {X 750.008,Y 2301.617,Z -203.448,A -89.15153,B 0.00000,C 180.00000} ; release
  LIN {X 750.008,Y 2301.617,Z 96.552,A -89.15153,B 0.00000,C 180.00000} ; retreat
  ; Step 1318, bar 2124
  LIN {X 1500.008,Y 2301.617,Z 992.570,A -89.15153,B 0.00000,C -180.00000} ; outside
  LIN {X 1500.008,Y 2301.617,Z 46.552,A -89.15153,B 0.00000,C -180.00000} ; preinsert
  LIN {X 1500.008,Y 2301.617,Z -203.448,A -89.15153,B 0.00000,C -180.00000} ; insert
  LIN {X 1500.008,Y 2301.617,Z -203.448,A -89.15153,B 0.00000,C -180.00000} ; release
  LIN {X 1500.008,Y 2301.617,Z 96.552,A -89.15153,B 0.00000,C -180.00000} ; retreat
  ; Step 1319, bar 2130
  LIN {X 2250.008,Y 2301.617,Z 992.570,A -89.15153,B 0.00000,C -180.00000} ; outside
  LIN {X 2250.008,Y 2301.617,Z 46.552,A -89.15153,B 0.00000,C -180.00000} ; preinsert
  LIN {X 2250.008,Y 2301.617,Z -203.448,A -89.15153,B 0.00000,C -180.00000} ; insert
  LIN {X 2250.008,Y 2301.617,Z -203.448,A -89.15153,B 0.00000,C -180.00000} ; release
  LIN {X 2250.008,Y 2301.617,Z 96.552,A -89.15153,B 0.00000,C -180.00000} ; retreat
  ; Step 1320, bar 2136
  LIN {X 3000.008,Y 2301.617,Z 992.570,A -89.15153,B 0.00000,C -180.00000} ; outside
  LIN {X 3000.008,Y 2301.617,Z 46.552,A -89.15153,B 0.00000,C -180.00000} ; preinsert
  LIN {X 3000.008,Y 2301.617,Z -203.448,A -89.15153,B 0.00000,C -180.00000} ; insert
  LIN {X 3000.008,Y 2301.617,Z -203.448,A -89.15153,B 0.00000,C -180.00000} ; release
  LIN {X 3000.008,Y 2301.617,Z 96.552,A -89.15153,B 0.00000,C -180.00000} ; retreat
  ; Step 1321, bar 2142
  LIN {X 3750.008,Y 2301.617,Z 992.570,A -89.15153,B 0.00000,C -180.00000} ; outside
  LIN {X 3750.008,Y 2301.617,Z 46.552,A -89.15153,B 0.00000,C -180.00000} ; preinsert
  LIN {X 3750.008,Y 2301.617,Z -203.448,A -89.15153,B 0.00000,C -180.00000} ; insert
  LIN {X 3750.008,Y 2301.617,Z -203.448,A -89.15153,B 0.00000,C -180.00000} ; release
  LIN {X 3750.008,Y 2301.617,Z 96.552,A -89.15153,B 0.00000,C -180.00000} ; retreat
  ; Step 1322, bar 2148
  LIN {X 4500.008,Y 2301.617,Z 992.570,A -89.15153,B 0.00000,C -180.00000} ; outside
  LIN {X 4500.008,Y 2301.617,Z 46.552,A -89.15153,B 0.00000,C -180.00000} ; preinsert
  LIN {X 4500.008,Y 2301.617,Z -203.448,A -89.15153,B 0.00000,C -180.00000} ; insert
  LIN {X 4500.008,Y 2301.617,Z -203.448,A -89.15153,B 0.00000,C -180.00000} ; release
  LIN {X 4500.008,Y 2301.617,Z 96.552,A -89.15153,B 0.00000,C -180.00000} ; retreat
  ; Step 1323, bar 2154
  LIN {X 5250.008,Y 2301.617,Z 992.570,A -89.15153,B 0.00000,C -180.00000} ; outside
  LIN {X 5250.008,Y 2301.617,Z 46.552,A -89.15153,B 0.00000,C -180.00000} ; preinsert
  LIN {X 5250.008,Y 2301.617,Z -203.448,A -89.15153,B 0.00000,C -180.00000} ; insert
  LIN {X 5250.008,Y 2301.617,Z -203.448,A -89.15153,B 0.00000,C -180.00000} ; release
  LIN {X 5250.008,Y 2301.617,Z 96.552,A -89.15153,B 0.00000,C -180.00000} ; retreat
  ; Step 1324, bar 2160
  LIN {X 6000.008,Y 2301.617,Z 992.570,A -89.15153,B 0.00000,C -180.00000} ; outside
  LIN {X 6000.008,Y 2301.617,Z 46.552,A -89.15153,B 0.00000,C -180.00000} ; preinsert
  LIN {X 6000.008,Y 2301.617,Z -203.448,A -89.15153,B 0.00000,C -180.00000} ; insert
  LIN {X 6000.008,Y 2301.617,Z -203.448,A -89.15153,B 0.00000,C -180.00000} ; release
  LIN {X 6000.008,Y 2301.617,Z 96.552,A -89.15153,B 0.00000,C -180.00000} ; retreat
  ; Step 1325, bar 2166
  LIN {X 6750.008,Y 2301.617,Z 992.570,A -89.15153,B 0.00000,C -180.00000} ; outside
  LIN {X 6750.008,Y 2301.617,Z 46.552,A -89.15153,B 0.00000,C -180.00000} ; preinsert
  LIN {X 6750.008,Y 2301.617,Z -203.448,A -89.15153,B 0.00000,C -180.00000} ; insert
  LIN {X 6750.008,Y 2301.617,Z -203.448,A -89.15153,B 0.00000,C -180.00000} ; release
  LIN {X 6750.008,Y 2301.617,Z 96.552,A -89.15153,B 0.00000,C -180.00000} ; retreat
  ; Step 1326, bar 2172
  LIN {X 7500.008,Y 2301.617,Z 992.570,A -89.15153,B 0.00000,C -180.00000} ; outside
  LIN {X 7500.008,Y 2301.617,Z 46.552,A -89.15153,B 0.00000,C -180.00000} ; preinsert
  LIN {X 7500.008,Y 2301.617,Z -203.448,A -89.15153,B 0.00000,C -180.00000} ; insert
  LIN {X 7500.008,Y 2301.617,Z -203.448,A -89.15153,B 0.00000,C -180.00000} ; release
  LIN {X 7500.008,Y 2301.617,Z 96.552,A -89.15153,B 0.00000,C -180.00000} ; retreat
  ; Step 1327, bar 2178
  LIN {X 8250.008,Y 2301.617,Z 992.570,A -89.15153,B 0.00000,C -180.00000} ; outside
  LIN {X 8250.008,Y 2301.617,Z 46.552,A -89.15153,B 0.00000,C -180.00000} ; preinsert
  LIN {X 8250.008,Y 2301.617,Z -203.448,A -89.15153,B 0.00000,C -180.00000} ; insert
  LIN {X 8250.008,Y 2301.617,Z -203.448,A -89.15153,B 0.00000,C -180.00000} ; release
  LIN {X 8250.008,Y 2301.617,Z 96.552,A -89.15153,B 0.00000,C -180.00000} ; retreat
  ; Step 1328, bar 2184
  LIN {X 9000.008,Y 2301.617,Z 992.570,A -89.15153,B 0.00000,C -180.00000} ; outside
  LIN {X 9000.008,Y 2301.617,Z 46.552,A -89.15153,B 0.00000,C -180.00000} ; preinsert
  LIN {X 9000.008,Y 2301.617,Z -203.448,A -89.15153,B 0.00000,C -180.00000} ; insert
  LIN {X 9000.008,Y 2301.617,Z -203.448,A -89.15153,B 0.00000,C -180.00000} ; release
  LIN {X 9000.008,Y 2301.617,Z 96.552,A -89.15153,B 0.00000,C -180.00000} ; retreat
  ; Step 1329, bar 2190
  LIN {X 9750.008,Y 2301.617,Z 992.570,A -89.15153,B 0.00000,C -180.00000} ; outside
  LIN {X 9750.008,Y 2301.617,Z 46.552,A -89.15153,B 0.00000,C -180.00000} ; preinsert
  LIN {X 9750.008,Y 2301.617,Z -203.448,A -89.15153,B 0.00000,C -180.00000} ; insert
  LIN {X 9750.008,Y 2301.617,Z -203.448,A -89.15153,B 0.00000,C -180.00000} ; release
  LIN {X 9750.008,Y 2301.617,Z 96.552,A -89.15153,B 0.00000,C -180.00000} ; retreat
  ; Step 1330, bar 2196
  LIN {X 10500.008,Y 2301.617,Z 992.570,A -89.15153,B 0.00000,C -180.00000} ; outside
  LIN {X 10500.008,Y 2301.617,Z 46.552,A -89.15153,B 0.00000,C -180.00000} ; preinsert
  LIN {X 10500.008,Y 2301.617,Z -203.448,A -89.15153,B 0.00000,C -180.00000} ; insert
  LIN {X 10500.008,Y 2301.617,Z -203.448,A -89.15153,B 0.00000,C -180.00000} ; release
  LIN {X 10500.008,Y 2301.617,Z 96.552,A -89.15153,B 0.00000,C -180.00000} ; retreat
  ; Step 1331, bar 2202
  LIN {X 11250.008,Y 2301.617,Z 992.570,A -89.15153,B 0.00000,C -180.00000} ; outside
  LIN {X 11250.008,Y 2301.617,Z 46.552,A -89.15153,B 0.00000,C -180.00000} ; preinsert
  LIN {X 11250.008,Y 2301.617,Z -203.448,A -89.15153,B 0.00000,C -180.00000} ; insert
  LIN {X 11250.008,Y 2301.617,Z -203.448,A -89.15153,B 0.00000,C -180.00000} ; release
  LIN {X 11250.008,Y 2301.617,Z 96.552,A -89.15153,B 0.00000,C -180.00000} ; retreat
  ; Step 1332, bar 2208
  LIN {X 12000.008,Y 2301.617,Z 992.570,A -89.15153,B 0.00000,C -180.00000} ; outside
  LIN {X 12000.008,Y 2301.617,Z 46.552,A -89.15153,B 0.00000,C -180.00000} ; preinsert
  LIN {X 12000.008,Y 2301.617,Z -203.448,A -89.15153,B 0.00000,C -180.00000} ; insert
  LIN {X 12000.008,Y 2301.617,Z -203.448,A -89.15153,B 0.00000,C -180.00000} ; release
  LIN {X 12000.008,Y 2301.617,Z 96.552,A -89.15153,B 0.00000,C -180.00000} ; retreat
  ; Step 1333, bar 2212
  LIN {X 12550.008,Y 2301.617,Z 992.570,A -89.15153,B 0.00000,C -180.00000} ; outside
  LIN {X 12550.008,Y 2301.617,Z 46.552,A -89.15153,B 0.00000,C -180.00000} ; preinsert
  LIN {X 12550.008,Y 2301.617,Z -203.448,A -89.15153,B 0.00000,C -180.00000} ; insert
  LIN {X 12550.008,Y 2301.617,Z -203.448,A -89.15153,B 0.00000,C -180.00000} ; release
  LIN {X 12550.008,Y 2301.617,Z 96.552,A -89.15153,B 0.00000,C -180.00000} ; retreat
  ; Step 1334, bar 2218
  LIN {X 13150.008,Y 2301.617,Z 992.570,A -89.15153,B 0.00000,C -180.00000} ; outside
  LIN {X 13150.008,Y 2301.617,Z 46.552,A -89.15153,B 0.00000,C -180.00000} ; preinsert
  LIN {X 13150.008,Y 2301.617,Z -203.448,A -89.15153,B 0.00000,C -180.00000} ; insert
  LIN {X 13150.008,Y 2301.617,Z -203.448,A -89.15153,B 0.00000,C -180.00000} ; release
  LIN {X 13150.008,Y 2301.617,Z 96.552,A -89.15153,B 0.00000,C -180.00000} ; retreat
  ; Step 1335, bar 2224
  LIN {X 13750.008,Y 2301.617,Z 992.570,A -89.15153,B 0.00000,C -180.00000} ; outside
  LIN {X 13750.008,Y 2301.617,Z 46.552,A -89.15153,B 0.00000,C -180.00000} ; preinsert
  LIN {X 13750.008,Y 2301.617,Z -203.448,A -89.15153,B 0.00000,C -180.00000} ; insert
  LIN {X 13750.008,Y 2301.617,Z -203.448,A -89.15153,B 0.00000,C -180.00000} ; release
  LIN {X 13750.008,Y 2301.617,Z 96.552,A -89.15153,B 0.00000,C -180.00000} ; retreat
  ; Step 1336, bar 2230
  LIN {X 14350.008,Y 2301.617,Z 992.570,A -89.15153,B 0.00000,C -180.00000} ; outside
  LIN {X 14350.008,Y 2301.617,Z 46.552,A -89.15153,B 0.00000,C -180.00000} ; preinsert
  LIN {X 14350.008,Y 2301.617,Z -203.448,A -89.15153,B 0.00000,C -180.00000} ; insert
  LIN {X 14350.008,Y 2301.617,Z -203.448,A -89.15153,B 0.00000,C -180.00000} ; release
  LIN {X 14350.008,Y 2301.617,Z 96.552,A -89.15153,B 0.00000,C -180.00000} ; retreat
  ; Step 1337, bar 2236
  LIN {X 14950.008,Y 2301.617,Z 992.570,A -89.15153,B 0.00000,C -180.00000} ; outside
  LIN {X 14950.008,Y 2301.617,Z 46.552,A -89.15153,B 0.00000,C -180.00000} ; preinsert
  LIN {X 14950.008,Y 2301.617,Z -203.448,A -89.15153,B 0.00000,C -180.00000} ; insert
  LIN {X 14950.008,Y 2301.617,Z -203.448,A -89.15153,B 0.00000,C -180.00000} ; release
  LIN {X 14950.008,Y 2301.617,Z 96.552,A -89.15153,B 0.00000,C -180.00000} ; retreat
  ; Step 1338, bar 2242
  LIN {X 15550.008,Y 2301.617,Z 992.570,A -89.15153,B 0.00000,C -180.00000} ; outside
  LIN {X 15550.008,Y 2301.617,Z 46.552,A -89.15153,B 0.00000,C -180.00000} ; preinsert
  LIN {X 15550.008,Y 2301.617,Z -203.448,A -89.15153,B 0.00000,C -180.00000} ; insert
  LIN {X 15550.008,Y 2301.617,Z -203.448,A -89.15153,B 0.00000,C -180.00000} ; release
  LIN {X 15550.008,Y 2301.617,Z 96.552,A -89.15153,B 0.00000,C -180.00000} ; retreat
  ; Step 1339, bar 2248
  LIN {X 16150.008,Y 2301.617,Z 992.570,A -89.15153,B 0.00000,C -180.00000} ; outside
  LIN {X 16150.008,Y 2301.617,Z 46.552,A -89.15153,B 0.00000,C -180.00000} ; preinsert
  LIN {X 16150.008,Y 2301.617,Z -203.448,A -89.15153,B 0.00000,C -180.00000} ; insert
  LIN {X 16150.008,Y 2301.617,Z -203.448,A -89.15153,B 0.00000,C -180.00000} ; release
  LIN {X 16150.008,Y 2301.617,Z 96.552,A -89.15153,B 0.00000,C -180.00000} ; retreat
  ; Step 1340, bar 1957
  LIN {X -13055.344,Y -1049.966,Z 919.196,A -179.99794,B 0.00000,C -180.00000} ; outside
  LIN {X -13055.344,Y -1049.966,Z -26.184,A -179.99794,B 0.00000,C -180.00000} ; preinsert
  LIN {X -13055.344,Y -1049.966,Z -276.184,A -179.99794,B 0.00000,C -180.00000} ; insert
  LIN {X -13055.344,Y -1049.966,Z -276.184,A -179.99794,B 0.00000,C -180.00000} ; release
  LIN {X -13055.344,Y -1049.966,Z 23.816,A -179.99794,B 0.00000,C -180.00000} ; retreat
  ; Step 1341, bar 1956
  LIN {X 13055.344,Y 1049.966,Z 919.196,A 0.00206,B 0.00000,C 180.00000} ; outside
  LIN {X 13055.344,Y 1049.966,Z -26.184,A 0.00206,B 0.00000,C 180.00000} ; preinsert
  LIN {X 13055.344,Y 1049.966,Z -276.184,A 0.00206,B 0.00000,C 180.00000} ; insert
  LIN {X 13055.344,Y 1049.966,Z -276.184,A 0.00206,B 0.00000,C 180.00000} ; release
  LIN {X 13055.344,Y 1049.966,Z 23.816,A 0.00206,B 0.00000,C 180.00000} ; retreat
  ; Step 1342, bar 1955
  LIN {X 13055.344,Y -1049.966,Z 919.196,A -0.00206,B 0.00000,C 180.00000} ; outside
  LIN {X 13055.344,Y -1049.966,Z -26.184,A -0.00206,B 0.00000,C 180.00000} ; preinsert
  LIN {X 13055.344,Y -1049.966,Z -276.184,A -0.00206,B 0.00000,C 180.00000} ; insert
  LIN {X 13055.344,Y -1049.966,Z -276.184,A -0.00206,B 0.00000,C 180.00000} ; release
  LIN {X 13055.344,Y -1049.966,Z 23.816,A -0.00206,B 0.00000,C 180.00000} ; retreat
  ; Step 1343, bar 1958
  LIN {X -13055.344,Y 1049.966,Z 919.196,A 179.99794,B 0.00000,C 180.00000} ; outside
  LIN {X -13055.344,Y 1049.966,Z -26.184,A 179.99794,B 0.00000,C 180.00000} ; preinsert
  LIN {X -13055.344,Y 1049.966,Z -276.184,A 179.99794,B 0.00000,C 180.00000} ; insert
  LIN {X -13055.344,Y 1049.966,Z -276.184,A 179.99794,B 0.00000,C 180.00000} ; release
  LIN {X -13055.344,Y 1049.966,Z 23.816,A 179.99794,B 0.00000,C 180.00000} ; retreat
  ; Step 1344, bar 2757
  LIN {X -1500.007,Y -1026.300,Z 1034.024,A 90.84369,B 0.00000,C 180.00000} ; outside
  LIN {X -1500.007,Y -1026.300,Z 88.277,A 90.84369,B 0.00000,C 180.00000} ; preinsert
  LIN {X -1500.007,Y -1026.300,Z -161.723,A 90.84369,B 0.00000,C 180.00000} ; insert
  LIN {X -1500.007,Y -1026.300,Z -161.723,A 90.84369,B 0.00000,C 180.00000} ; release
  LIN {X -1500.007,Y -1026.300,Z 138.277,A 90.84369,B 0.00000,C 180.00000} ; retreat
  ; Step 1345, bar 2754
  LIN {X -750.007,Y -1026.300,Z 1034.024,A 90.84369,B 0.00000,C 180.00000} ; outside
  LIN {X -750.007,Y -1026.300,Z 88.277,A 90.84369,B 0.00000,C 180.00000} ; preinsert
  LIN {X -750.007,Y -1026.300,Z -161.723,A 90.84369,B 0.00000,C 180.00000} ; insert
  LIN {X -750.007,Y -1026.300,Z -161.723,A 90.84369,B 0.00000,C 180.00000} ; release
  LIN {X -750.007,Y -1026.300,Z 138.277,A 90.84369,B 0.00000,C 180.00000} ; retreat
  ; Step 1346, bar 2751
  LIN {X -0.007,Y -1026.300,Z 1034.024,A 90.84369,B 0.00000,C -180.00000} ; outside
  LIN {X -0.007,Y -1026.300,Z 88.277,A 90.84369,B 0.00000,C -180.00000} ; preinsert
  LIN {X -0.007,Y -1026.300,Z -161.723,A 90.84369,B 0.00000,C -180.00000} ; insert
  LIN {X -0.007,Y -1026.300,Z -161.723,A 90.84369,B 0.00000,C -180.00000} ; release
  LIN {X -0.007,Y -1026.300,Z 138.277,A 90.84369,B 0.00000,C -180.00000} ; retreat
  ; Step 1347, bar 2802
  LIN {X 750.007,Y -1026.300,Z 1034.024,A 89.15631,B 0.00000,C 180.00000} ; outside
  LIN {X 750.007,Y -1026.300,Z 88.277,A 89.15631,B 0.00000,C 180.00000} ; preinsert
  LIN {X 750.007,Y -1026.300,Z -161.723,A 89.15631,B 0.00000,C 180.00000} ; insert
  LIN {X 750.007,Y -1026.300,Z -161.723,A 89.15631,B 0.00000,C 180.00000} ; release
  LIN {X 750.007,Y -1026.300,Z 138.277,A 89.15631,B 0.00000,C 180.00000} ; retreat
  ; Step 1348, bar 2805
  LIN {X 1500.007,Y -1026.300,Z 1034.024,A 89.15631,B 0.00000,C -180.00000} ; outside
  LIN {X 1500.007,Y -1026.300,Z 88.277,A 89.15631,B 0.00000,C -180.00000} ; preinsert
  LIN {X 1500.007,Y -1026.300,Z -161.723,A 89.15631,B 0.00000,C -180.00000} ; insert
  LIN {X 1500.007,Y -1026.300,Z -161.723,A 89.15631,B 0.00000,C -180.00000} ; release
  LIN {X 1500.007,Y -1026.300,Z 138.277,A 89.15631,B 0.00000,C -180.00000} ; retreat
  ; Step 1349, bar 2808
  LIN {X 2250.007,Y -1026.300,Z 1034.024,A 89.15631,B 0.00000,C 180.00000} ; outside
  LIN {X 2250.007,Y -1026.300,Z 88.277,A 89.15631,B 0.00000,C 180.00000} ; preinsert
  LIN {X 2250.007,Y -1026.300,Z -161.723,A 89.15631,B 0.00000,C 180.00000} ; insert
  LIN {X 2250.007,Y -1026.300,Z -161.723,A 89.15631,B 0.00000,C 180.00000} ; release
  LIN {X 2250.007,Y -1026.300,Z 138.277,A 89.15631,B 0.00000,C 180.00000} ; retreat
  ; Step 1350, bar 2811
  LIN {X 3000.007,Y -1026.300,Z 1034.024,A 89.15631,B 0.00000,C 180.00000} ; outside
  LIN {X 3000.007,Y -1026.300,Z 88.277,A 89.15631,B 0.00000,C 180.00000} ; preinsert
  LIN {X 3000.007,Y -1026.300,Z -161.723,A 89.15631,B 0.00000,C 180.00000} ; insert
